C07295=1140.196,8.392,-49.288,179.724,6.289,149.221
C07296=1140.191,8.641,-49.301,179.727,6.291,149.220
C07297=1140.186,8.891,-49.315,179.729,6.291,149.220
C07298=1140.180,9.141,-49.329,179.732,6.292,149.219
C07299=1140.176,9.390,-49.342,179.734,6.293,149.219
C07300=1140.170,9.640,-49.355,179.737,6.294,149.218
C07301=1140.165,9.889,-49.370,179.739,6.295,149.218
C07302=1140.160,10.139,-49.382,179.741,6.296,149.217
C07303=1140.155,10.388,-49.397,179.744,6.296,149.216
C07304=1140.150,10.639,-49.410,179.747,6.298,149.216
C07305=1140.145,10.887,-49.423,179.749,6.298,149.215
C07306=1140.140,11.137,-49.438,179.752,6.299,149.215
C07307=1140.134,11.387,-49.451,179.754,6.300,149.214
C07308=1140.129,11.636,-49.465,179.757,6.301,149.214
C07309=1140.125,11.886,-49.478,179.759,6.302,149.213
C07310=1140.119,12.136,-49.492,179.762,6.303,149.213
C07311=1140.114,12.385,-49.506,179.765,6.304,149.212
C07312=1140.109,12.635,-49.520,179.767,6.305,149.212
C07313=1140.104,12.884,-49.533,179.770,6.305,149.211
C07314=1140.099,13.134,-49.547,179.772,6.306,149.210
C07315=1140.094,13.384,-49.561,179.775,6.307,149.210
C07316=1140.089,13.633,-49.575,179.777,6.308,149.209
C07317=1140.084,13.882,-49.588,179.779,6.309,149.209
C07318=1140.078,14.132,-49.602,179.782,6.310,149.208
C07319=1140.074,14.382,-49.616,179.785,6.311,149.208
C07320=1140.068,14.631,-49.630,179.787,6.312,149.207
C07321=1140.063,14.881,-49.644,179.790,6.312,149.207
C07322=1140.058,15.131,-49.657,179.792,6.314,149.206
C07323=1140.053,15.380,-49.671,179.795,6.314,149.206
C07324=1140.048,15.629,-49.685,179.797,6.315,149.205
C07325=1140.042,15.878,-49.699,179.800,6.316,149.204
C07326=1140.037,16.129,-49.713,179.802,6.317,149.204
C07327=1140.033,16.378,-49.727,179.805,6.318,149.203
C07328=1140.027,16.627,-49.741,179.808,6.319,149.203
C07329=1140.022,16.877,-49.755,179.810,6.320,149.202
C07330=1140.017,17.127,-49.769,179.812,6.321,149.202
C07331=1140.012,17.377,-49.783,179.815,6.322,149.201
C07332=1140.007,17.626,-49.797,179.818,6.323,149.201
C07333=1140.002,17.876,-49.811,179.820,6.323,149.200
C07334=1139.997,18.125,-49.825,179.823,6.325,149.199
C07335=1139.992,18.374,-49.838,179.825,6.326,149.199
C07336=1139.987,18.624,-49.853,179.828,6.326,149.199
C07337=1139.982,18.874,-49.866,179.830,6.327,149.198
C07338=1139.976,19.123,-49.880,179.833,6.328,149.197
C07339=1139.971,19.373,-49.894,179.835,6.329,149.197
C07340=1139.966,19.623,-49.909,179.838,6.330,149.196
C07341=1139.961,19.872,-49.923,179.841,6.331,149.196
C07342=1139.956,20.121,-49.937,179.843,6.332,149.195
C07343=1139.951,20.371,-49.951,179.845,6.333,149.195
C07344=1139.946,20.621,-49.965,179.848,6.334,149.194
C07345=1139.940,20.870,-49.979,179.851,6.335,149.194
C07346=1139.935,21.119,-49.994,179.854,6.336,149.193
C07347=1139.930,21.369,-50.008,179.856,6.337,149.193
C07348=1139.925,21.619,-50.022,179.858,6.337,149.192
C07349=1139.920,21.869,-50.037,179.861,6.339,149.191
C07350=1139.915,22.118,-50.050,179.864,6.340,149.191
C07351=1139.910,22.367,-50.065,179.866,6.340,149.190
C07352=1139.905,22.617,-50.079,179.869,6.342,149.190
C07353=1139.900,22.867,-50.093,179.871,6.342,149.189
C07354=1139.894,23.116,-50.107,179.874,6.343,149.189
C07355=1139.890,23.365,-50.121,179.876,6.345,149.188
C07356=1139.885,23.615,-50.136,179.879,6.345,149.188
C07357=1139.880,23.865,-50.150,179.881,6.346,149.187
C07358=1139.875,24.115,-50.164,179.884,6.347,149.186
C07359=1139.869,24.364,-50.178,179.887,6.348,149.186
C07360=1139.864,24.613,-50.192,179.889,6.349,149.186
C07361=1139.859,24.863,-50.207,179.892,6.350,149.185
C07362=1139.854,25.113,-50.221,179.894,6.351,149.184
C07363=1139.849,25.362,-50.235,179.897,6.353,149.184
C07364=1139.844,25.611,-50.249,179.900,6.353,149.183
C07365=1139.839,25.861,-50.264,179.902,6.354,149.183
C07366=1139.834,26.110,-50.278,179.905,6.355,149.182
C07367=1139.829,26.360,-50.293,179.907,6.356,149.182
C07368=1139.824,26.610,-50.307,179.909,6.357,149.181
C07369=1139.819,26.859,-50.321,179.913,6.358,149.181
C07370=1139.813,27.128,-50.337,179.915,6.359,149.180
C07371=1139.807,27.397,-50.352,179.918,6.360,149.179
C07372=1139.802,27.666,-50.368,179.921,6.362,149.179
C07373=1139.797,27.935,-50.384,179.923,6.362,149.178
C07374=1139.791,28.185,-50.399,179.926,6.363,149.178
C07375=1139.786,28.435,-50.413,179.929,6.364,149.177
C07376=1139.782,28.684,-50.427,179.931,6.365,149.177
C07377=1139.777,28.933,-50.442,179.934,6.367,149.176
C07378=1139.771,29.182,-50.456,179.936,6.367,149.176
C07379=1139.766,29.432,-50.470,179.939,6.368,149.175
C07380=1139.761,29.682,-50.485,179.941,6.370,149.175
C07381=1139.756,29.931,-50.500,179.944,6.370,149.174
C07382=1139.751,30.181,-50.514,179.947,6.372,149.174
C07383=1139.746,30.431,-50.529,179.949,6.373,149.173
C07384=1139.741,30.680,-50.544,179.952,6.373,149.172
C07385=1139.737,30.929,-50.558,179.954,6.375,149.172
C07386=1139.731,31.179,-50.573,179.957,6.375,149.171
C07387=1139.726,31.428,-50.588,179.960,6.377,149.171
C07388=1139.721,31.678,-50.602,179.962,6.378,149.170
C07389=1139.716,31.927,-50.616,179.965,6.379,149.170
C07390=1139.710,32.177,-50.632,179.967,6.380,149.169
C07391=1139.705,32.426,-50.646,179.969,6.380,149.169
C07392=1139.700,32.676,-50.660,179.973,6.382,149.168
C07393=1139.696,32.925,-50.675,179.975,6.383,149.168
C07394=1139.690,33.175,-50.690,179.978,6.384,149.167
C07395=1139.685,33.424,-50.705,179.980,6.385,149.167
C07396=1139.680,33.674,-50.719,179.982,6.385,149.166
C07397=1139.675,33.924,-50.734,179.986,6.387,149.165
C07398=1139.670,34.173,-50.749,179.988,6.387,149.165
C07399=1139.665,34.423,-50.763,179.991,6.389,149.165
C07400=1139.660,34.672,-50.778,179.993,6.390,149.164
C07401=1139.655,34.922,-50.793,179.996,6.391,149.163
C07402=1139.650,35.171,-50.808,179.998,6.392,149.163
C07403=1139.645,35.421,-50.823,-179.999,6.393,149.162
C07404=1139.640,35.670,-50.838,-179.996,6.394,149.162
C07405=1139.635,35.920,-50.852,-179.994,6.395,149.161
C07406=1139.630,36.169,-50.867,-179.991,6.396,149.161
C07407=1139.624,36.419,-50.882,-179.989,6.397,149.160
C07408=1139.620,36.668,-50.897,-179.986,6.399,149.160
C07409=1139.614,36.918,-50.912,-179.983,6.399,149.159
C07410=1139.609,37.167,-50.927,-179.981,6.401,149.159
C07411=1139.605,37.417,-50.941,-179.978,6.401,149.158
C07412=1139.599,37.666,-50.957,-179.975,6.403,149.158
C07413=1139.594,37.916,-50.971,-179.973,6.404,149.157
C07414=1139.589,38.165,-50.987,-179.970,6.404,149.156
C07415=1139.584,38.414,-51.002,-179.968,6.406,149.156
C07416=1139.579,38.664,-51.016,-179.965,6.407,149.156
C07417=1139.574,38.914,-51.032,-179.962,6.408,149.155
C07418=1139.569,39.163,-51.046,-179.960,6.409,149.154
C07419=1139.563,39.413,-51.062,-179.957,6.410,149.154
C07420=1139.559,39.662,-51.077,-179.955,6.411,149.153
C07421=1139.553,39.912,-51.091,-179.952,6.412,149.153
C07422=1139.549,40.162,-51.107,-179.950,6.413,149.152
C07423=1139.544,40.411,-51.122,-179.947,6.414,149.152
C07424=1139.539,40.661,-51.137,-179.944,6.415,149.151
C07425=1139.534,40.910,-51.152,-179.942,6.417,149.151
C07426=1139.529,41.159,-51.167,-179.939,6.417,149.150
C07427=1139.524,41.409,-51.182,-179.936,6.419,149.150
C07428=1139.518,41.658,-51.197,-179.934,6.420,149.149
C07429=1139.514,41.907,-51.212,-179.931,6.421,149.149
C07430=1139.508,42.157,-51.228,-179.929,6.422,149.148
C07431=1139.503,42.406,-51.242,-179.926,6.424,149.148
C07432=1139.498,42.656,-51.258,-179.923,6.424,149.147
C07433=1139.494,42.906,-51.273,-179.920,6.426,149.147
C07434=1139.489,43.155,-51.289,-179.918,6.426,149.146
C07435=1139.483,43.405,-51.303,-179.915,6.428,149.145
C07436=1139.478,43.654,-51.318,-179.913,6.429,149.145
C07437=1139.473,43.904,-51.334,-179.910,6.430,149.144
C07438=1139.468,44.153,-51.349,-179.907,6.431,149.144
C07439=1139.463,44.402,-51.365,-179.905,6.432,149.143
C07440=1139.459,44.652,-51.380,-179.902,6.433,149.143
C07441=1139.453,44.902,-51.395,-179.899,6.434,149.142
C07442=1139.448,45.151,-51.410,-179.897,6.435,149.142
C07443=1139.443,45.400,-51.425,-179.894,6.436,149.141
C07444=1139.438,45.650,-51.441,-179.892,6.437,149.141
C07445=1139.433,45.899,-51.456,-179.889,6.439,149.140
C07446=1139.428,46.149,-51.472,-179.886,6.439,149.140
C07447=1139.423,46.398,-51.487,-179.884,6.441,149.139
C07448=1139.418,46.647,-51.502,-179.881,6.442,149.139
C07449=1139.412,46.897,-51.517,-179.878,6.443,149.138
C07450=1139.408,47.147,-51.532,-179.876,6.444,149.138
C07451=1139.403,47.397,-51.548,-179.873,6.446,149.137
C07452=1139.398,47.646,-51.564,-179.871,6.446,149.136
C07453=1139.393,47.895,-51.579,-179.868,6.448,149.136
C07454=1139.388,48.145,-51.594,-179.866,6.449,149.136
C07455=1139.383,48.395,-51.610,-179.862,6.450,149.135
C07456=1139.378,48.644,-51.625,-179.860,6.451,149.134
C07457=1139.373,48.893,-51.641,-179.858,6.452,149.134
C07458=1139.367,49.143,-51.657,-179.855,6.453,149.134
C07459=1139.363,49.392,-51.672,-179.852,6.454,149.133
C07460=1139.358,49.642,-51.688,-179.849,6.456,149.132
C07461=1139.353,49.891,-51.703,-179.847,6.457,149.132
C07462=1139.347,50.141,-51.719,-179.844,6.458,149.131
C07463=1139.343,50.390,-51.734,-179.842,6.459,149.131
C07464=1139.338,50.640,-51.750,-179.839,6.461,149.130
C07465=1139.333,50.889,-51.766,-179.836,6.461,149.130
C07466=1139.327,51.138,-51.782,-179.834,6.463,149.129
C07467=1139.323,51.388,-51.797,-179.832,6.464,149.129
C07468=1139.318,51.637,-51.812,-179.828,6.465,149.128
C07469=1139.312,51.887,-51.828,-179.826,6.466,149.128
C07470=1139.307,52.136,-51.844,-179.823,6.467,149.127
C07471=1139.303,52.386,-51.859,-179.820,6.469,149.127
C07472=1139.298,52.635,-51.875,-179.818,6.469,149.126
C07473=1139.292,52.885,-51.890,-179.815,6.471,149.126
C07474=1139.287,53.153,-51.907,-179.813,6.472,149.125
C07475=1139.282,53.422,-51.925,-179.810,6.473,149.125
C07476=1139.276,53.691,-51.942,-179.807,6.474,149.124
C07477=1139.271,53.959,-51.958,-179.804,6.476,149.124
C07478=1139.266,54.208,-51.974,-179.801,6.477,149.123
C07479=1139.261,54.458,-51.990,-179.798,6.478,149.122
C07480=1139.256,54.707,-52.006,-179.796,6.479,149.122
C07481=1139.251,54.957,-52.021,-179.793,6.480,149.121
C07482=1139.246,55.207,-52.037,-179.790,6.482,149.121
C07483=1139.241,55.456,-52.053,-179.788,6.483,149.120
C07484=1139.235,55.705,-52.069,-179.785,6.484,149.120
C07485=1139.231,55.955,-52.085,-179.783,6.485,149.119
C07486=1139.226,56.204,-52.100,-179.780,6.487,149.119
C07487=1139.221,56.453,-52.117,-179.777,6.488,149.119
C07488=1139.216,56.703,-52.133,-179.775,6.489,149.118
C07489=1139.211,56.952,-52.148,-179.772,6.490,149.117
C07490=1139.206,57.202,-52.164,-179.770,6.491,149.117
C07491=1139.201,57.451,-52.180,-179.766,6.492,149.116
C07492=1139.196,57.701,-52.196,-179.764,6.494,149.116
C07493=1139.191,57.951,-52.212,-179.762,6.495,149.115
C07494=1139.186,58.200,-52.228,-179.758,6.496,149.115
C07495=1139.180,58.449,-52.244,-179.756,6.497,149.114
C07496=1139.176,58.698,-52.260,-179.753,6.499,149.114
C07497=1139.170,58.948,-52.276,-179.751,6.500,149.113
C07498=1139.166,59.198,-52.292,-179.748,6.501,149.113
C07499=1139.161,59.446,-52.308,-179.745,6.502,149.112
C07500=1139.156,59.696,-52.324,-179.743,6.503,149.112
C07501=1139.151,59.945,-52.340,-179.740,6.505,149.111
C07502=1139.146,60.195,-52.356,-179.737,6.506,149.111
C07503=1139.142,60.444,-52.372,-179.735,6.507,149.110
C07504=1139.136,60.694,-52.388,-179.732,6.508,149.110
C07505=1139.131,60.944,-52.404,-179.729,6.510,149.109
C07506=1139.126,61.193,-52.421,-179.727,6.511,149.109
C07507=1139.121,61.443,-52.437,-179.724,6.512,149.108
C07508=1139.116,61.692,-52.453,-179.721,6.513,149.108
C07509=1139.111,61.942,-52.469,-179.719,6.515,149.107
C07510=1139.106,62.191,-52.485,-179.716,6.516,149.107
C07511=1139.101,62.441,-52.501,-179.713,6.517,149.106
C07512=1139.096,62.689,-52.517,-179.711,6.518,149.106
C07513=1139.091,62.939,-52.534,-179.708,6.520,149.105
C07514=1139.086,63.188,-52.550,-179.706,6.521,149.105
C07515=1139.082,63.438,-52.566,-179.702,6.522,149.104
C07516=1139.076,63.687,-52.582,-179.700,6.523,149.104
C07517=1139.072,63.937,-52.599,-179.697,6.525,149.103
C07518=1139.066,64.186,-52.614,-179.694,6.526,149.103
C07519=1139.062,64.436,-52.631,-179.692,6.527,149.102
C07520=1139.056,64.685,-52.648,-179.689,6.528,149.102
C07521=1139.051,64.935,-52.664,-179.687,6.530,149.101
C07522=1139.046,65.184,-52.680,-179.684,6.530,149.101
C07523=1139.042,65.433,-52.697,-179.681,6.532,149.100
C07524=1139.036,65.682,-52.712,-179.678,6.534,149.100
C07525=1139.032,65.932,-52.729,-179.676,6.534,149.099
C07526=1139.027,66.181,-52.745,-179.673,6.536,149.099
C07527=1139.021,66.431,-52.762,-179.670,6.538,149.098
C07528=1139.016,66.680,-52.778,-179.668,6.538,149.098
C07529=1139.012,66.929,-52.795,-179.665,6.540,149.097
C07530=1139.007,67.179,-52.811,-179.662,6.541,149.097
C07531=1139.002,67.428,-52.827,-179.660,6.542,149.096
C07532=1138.997,67.678,-52.844,-179.657,6.544,149.096
C07533=1138.992,67.927,-52.861,-179.654,6.545,149.095
C07534=1138.987,68.177,-52.877,-179.652,6.546,149.095
C07535=1138.982,68.426,-52.893,-179.649,6.548,149.094
C07536=1138.977,68.675,-52.910,-179.646,6.549,149.094
C07537=1138.972,68.925,-52.927,-179.644,6.550,149.093
C07538=1138.967,69.174,-52.943,-179.641,6.551,149.093
C07539=1138.962,69.424,-52.959,-179.638,6.553,149.092
C07540=1138.957,69.673,-52.975,-179.636,6.553,149.092
C07541=1138.952,69.922,-52.993,-179.633,6.555,149.091
C07542=1138.947,70.172,-53.009,-179.630,6.557,149.091
C07543=1138.942,70.421,-53.026,-179.627,6.558,149.090
C07544=1138.938,70.670,-53.042,-179.625,6.559,149.090
C07545=1138.933,70.920,-53.060,-179.622,6.561,149.089
C07546=1138.927,71.169,-53.075,-179.619,6.562,149.089
C07547=1138.923,71.419,-53.092,-179.617,6.563,149.088
C07548=1138.917,71.669,-53.109,-179.614,6.564,149.088
C07549=1138.912,71.917,-53.125,-179.611,6.566,149.087
C07550=1138.908,72.167,-53.142,-179.609,6.567,149.087
C07551=1138.902,72.416,-53.159,-179.606,6.569,149.087
C07552=1138.898,72.666,-53.176,-179.603,6.570,149.086
C07553=1138.893,72.915,-53.192,-179.600,6.571,149.085
C07554=1138.887,73.164,-53.209,-179.598,6.572,149.085
C07555=1138.883,73.414,-53.226,-179.595,6.574,149.085
C07556=1138.878,73.663,-53.242,-179.592,6.575,149.084
C07557=1138.873,73.913,-53.260,-179.590,6.576,149.083
C07558=1138.868,74.162,-53.276,-179.587,6.578,149.083
C07559=1138.863,74.411,-53.293,-179.584,6.579,149.082
C07560=1138.858,74.661,-53.310,-179.581,6.581,149.082
C07561=1138.853,74.910,-53.326,-179.579,6.582,149.082
C07562=1138.848,75.160,-53.344,-179.576,6.583,149.081
C07563=1138.844,75.409,-53.360,-179.574,6.585,149.081
C07564=1138.838,75.659,-53.377,-179.571,6.585,149.080
C07565=1138.833,75.908,-53.394,-179.568,6.587,149.080
C07566=1138.828,76.157,-53.411,-179.566,6.589,149.079
C07567=1138.824,76.407,-53.428,-179.563,6.590,149.079
C07568=1138.818,76.656,-53.445,-179.560,6.591,149.078
C07569=1138.814,76.905,-53.462,-179.557,6.592,149.078
C07570=1138.809,77.154,-53.479,-179.555,6.594,149.077
C07571=1138.804,77.404,-53.496,-179.552,6.596,149.077
C07572=1138.799,77.653,-53.512,-179.549,6.596,149.076
C07573=1138.794,77.903,-53.530,-179.547,6.598,149.076
C07574=1138.789,78.152,-53.546,-179.544,6.600,149.075
C07575=1138.784,78.402,-53.563,-179.541,6.601,149.075
C07576=1138.780,78.651,-53.581,-179.538,6.602,149.074
C07577=1138.774,78.900,-53.598,-179.536,6.603,149.074
C07578=1138.768,79.169,-53.616,-179.533,6.605,149.073
C07579=1138.763,79.437,-53.634,-179.530,6.606,149.073
C07580=1138.758,79.706,-53.653,-179.527,6.608,149.072
C07581=1138.753,79.974,-53.671,-179.524,6.610,149.072
C07582=1138.748,80.224,-53.688,-179.521,6.611,149.071
C07583=1138.742,80.472,-53.706,-179.518,6.613,149.071
C07584=1138.738,80.722,-53.723,-179.516,6.613,149.070
C07585=1138.733,80.972,-53.740,-179.513,6.615,149.070
C07586=1138.729,81.220,-53.757,-179.510,6.616,149.069
C07587=1138.723,81.470,-53.774,-179.507,6.618,149.069
C07588=1138.718,81.719,-53.791,-179.505,6.619,149.068
C07589=1138.713,81.968,-53.809,-179.502,6.621,149.068
C07590=1138.708,82.218,-53.826,-179.500,6.622,149.068
C07591=1138.704,82.468,-53.843,-179.497,6.624,149.067
C07592=1138.699,82.717,-53.861,-179.494,6.625,149.066
C07593=1138.694,82.966,-53.878,-179.492,6.626,149.066
C07594=1138.689,83.216,-53.895,-179.489,6.628,149.066
C07595=1138.684,83.464,-53.912,-179.486,6.629,149.065
C07596=1138.678,83.714,-53.929,-179.483,6.631,149.065
C07597=1138.674,83.963,-53.947,-179.480,6.632,149.064
C07598=1138.669,84.213,-53.964,-179.478,6.633,149.064
C07599=1138.664,84.463,-53.981,-179.475,6.635,149.063
C07600=1138.660,84.712,-53.999,-179.472,6.636,149.063
C07601=1138.654,84.961,-54.016,-179.469,6.638,149.062
C07602=1138.649,85.211,-54.034,-179.467,6.639,149.062
C07603=1138.645,85.460,-54.051,-179.464,6.640,149.061
C07604=1138.639,85.708,-54.068,-179.462,6.642,149.061
C07605=1138.634,85.958,-54.086,-179.458,6.643,149.060
C07606=1138.629,86.207,-54.103,-179.456,6.645,149.060
C07607=1138.625,86.457,-54.120,-179.453,6.647,149.059
C07608=1138.620,86.706,-54.138,-179.451,6.647,149.059
C07609=1138.615,86.956,-54.155,-179.448,6.649,149.059
C07610=1138.610,87.205,-54.173,-179.445,6.650,149.058
C07611=1138.605,87.455,-54.190,-179.442,6.652,149.057
C07612=1138.600,87.704,-54.208,-179.439,6.654,149.057
C07613=1138.595,87.953,-54.226,-179.437,6.655,149.057
C07614=1138.590,88.203,-54.243,-179.434,6.656,149.056
C07615=1138.585,88.452,-54.261,-179.431,6.658,149.056
C07616=1138.581,88.701,-54.278,-179.429,6.659,149.055
C07617=1138.576,88.951,-54.296,-179.426,6.661,149.055
C07618=1138.571,89.200,-54.314,-179.423,6.663,149.054
C07619=1138.566,89.450,-54.331,-179.421,6.663,149.054
C07620=1138.561,89.699,-54.349,-179.418,6.665,149.053
C07621=1138.557,89.948,-54.367,-179.415,6.666,149.053
C07622=1138.552,90.197,-54.384,-179.412,6.668,149.052
C07623=1138.547,90.447,-54.402,-179.409,6.670,149.052
C07624=1138.542,90.696,-54.420,-179.407,6.671,149.052
C07625=1138.536,90.946,-54.437,-179.404,6.673,149.051
C07626=1138.532,91.195,-54.455,-179.401,6.674,149.050
C07627=1138.527,91.444,-54.473,-179.399,6.675,149.050
C07628=1138.522,91.693,-54.491,-179.396,6.677,149.050
C07629=1138.517,91.943,-54.508,-179.393,6.679,149.049
C07630=1138.512,92.192,-54.526,-179.390,6.680,149.049
C07631=1138.507,92.441,-54.544,-179.388,6.682,149.048
C07632=1138.503,92.690,-54.562,-179.385,6.682,149.048
C07633=1138.497,92.940,-54.579,-179.382,6.684,149.047
C07634=1138.492,93.189,-54.597,-179.380,6.686,149.047
C07635=1138.487,93.438,-54.615,-179.377,6.687,149.046
C07636=1138.483,93.687,-54.633,-179.374,6.689,149.046
C07637=1138.478,93.937,-54.651,-179.371,6.691,149.046
C07638=1138.473,94.186,-54.669,-179.368,6.692,149.045
C07639=1138.468,94.436,-54.686,-179.365,6.694,149.045
C07640=1138.463,94.685,-54.704,-179.363,6.695,149.044
C07641=1138.458,94.935,-54.722,-179.361,6.696,149.044
C07642=1138.453,95.184,-54.740,-179.358,6.698,149.043
C07643=1138.448,95.433,-54.758,-179.355,6.700,149.043
C07644=1138.444,95.682,-54.776,-179.352,6.701,149.042
C07645=1138.439,95.931,-54.794,-179.349,6.703,149.042
C07646=1138.434,96.180,-54.812,-179.346,6.704,149.041
C07647=1138.429,96.430,-54.830,-179.344,6.706,149.041
C07648=1138.424,96.679,-54.848,-179.341,6.708,149.041
C07649=1138.419,96.928,-54.866,-179.339,6.708,149.040
C07650=1138.415,97.178,-54.884,-179.336,6.710,149.039
C07651=1138.410,97.427,-54.902,-179.333,6.711,149.039
C07652=1138.405,97.676,-54.920,-179.330,6.713,149.039
C07653=1138.400,97.925,-54.938,-179.327,6.715,149.038
C07654=1138.395,98.175,-54.956,-179.325,6.716,149.038
C07655=1138.390,98.424,-54.974,-179.322,6.718,149.037
C07656=1138.384,98.673,-54.993,-179.319,6.720,149.037
C07657=1138.380,98.923,-55.011,-179.316,6.721,149.036
C07658=1138.375,99.172,-55.029,-179.313,6.723,149.036
C07659=1138.370,99.421,-55.047,-179.311,6.724,149.036
C07660=1138.365,99.671,-55.065,-179.308,6.725,149.035
C07661=1138.361,99.920,-55.083,-179.306,6.727,149.035
C07662=1138.356,100.169,-55.101,-179.303,6.729,149.034
C07663=1138.351,100.419,-55.120,-179.300,6.730,149.034
C07664=1138.346,100.668,-55.138,-179.297,6.732,149.033
C07665=1138.341,100.918,-55.156,-179.294,6.733,149.033
C07666=1138.336,101.166,-55.175,-179.291,6.735,149.032
C07667=1138.331,101.415,-55.193,-179.289,6.737,149.032
C07668=1138.327,101.665,-55.211,-179.286,6.738,149.032
C07669=1138.321,101.915,-55.230,-179.283,6.740,149.031
C07670=1138.316,102.164,-55.248,-179.280,6.742,149.031
C07671=1138.311,102.413,-55.266,-179.278,6.743,149.030
C07672=1138.307,102.662,-55.285,-179.275,6.744,149.030
C07673=1138.303,102.911,-55.303,-179.272,6.746,149.029
C07674=1138.297,103.161,-55.321,-179.270,6.747,149.029
C07675=1138.292,103.410,-55.339,-179.267,6.749,149.028
C07676=1138.288,103.659,-55.358,-179.264,6.751,149.028
C07677=1138.283,103.908,-55.376,-179.261,6.752,149.028
C07678=1138.277,104.158,-55.395,-179.259,6.754,149.027
C07679=1138.272,104.407,-55.413,-179.256,6.756,149.027
C07680=1138.268,104.656,-55.432,-179.253,6.757,149.026
C07681=1138.264,104.906,-55.450,-179.250,6.759,149.026
C07682=1138.258,105.174,-55.470,-179.247,6.760,149.025
C07683=1138.253,105.442,-55.490,-179.245,6.762,149.025
C07684=1138.248,105.711,-55.510,-179.241,6.764,149.024
C07685=1138.243,105.979,-55.530,-179.238,6.766,149.024
C07686=1138.237,106.229,-55.548,-179.235,6.767,149.023
C07687=1138.232,106.477,-55.567,-179.232,6.769,149.023
C07688=1138.228,106.727,-55.585,-179.230,6.771,149.023
C07689=1138.223,106.976,-55.605,-179.227,6.772,149.022
C07690=1138.218,107.225,-55.623,-179.224,6.774,149.022
C07691=1138.214,107.475,-55.641,-179.222,6.776,149.021
C07692=1138.208,107.724,-55.660,-179.219,6.777,149.021
C07693=1138.203,107.973,-55.678,-179.217,6.778,149.021
C07694=1138.199,108.222,-55.697,-179.213,6.780,149.020
C07695=1138.194,108.472,-55.716,-179.211,6.781,149.020
C07696=1138.189,108.720,-55.735,-179.208,6.783,149.019
C07697=1138.184,108.971,-55.754,-179.205,6.785,149.019
C07698=1138.179,109.219,-55.772,-179.203,6.786,149.018
C07699=1138.174,109.469,-55.791,-179.200,6.788,149.018
C07700=1138.170,109.718,-55.810,-179.197,6.790,149.017
C07701=1138.165,109.967,-55.828,-179.194,6.791,149.017
C07702=1138.160,110.217,-55.848,-179.192,6.793,149.017
C07703=1138.155,110.466,-55.866,-179.189,6.795,149.016
C07704=1138.150,110.715,-55.885,-179.186,6.796,149.016
C07705=1138.146,110.964,-55.904,-179.183,6.798,149.015
C07706=1138.140,111.214,-55.922,-179.180,6.799,149.015
C07707=1138.136,111.463,-55.942,-179.177,6.801,149.014
C07708=1138.130,111.712,-55.960,-179.175,6.803,149.014
C07709=1138.126,111.961,-55.979,-179.172,6.805,149.014
C07710=1138.121,112.210,-55.998,-179.169,6.806,149.013
C07711=1138.116,112.460,-56.016,-179.167,6.808,149.013
C07712=1138.111,112.709,-56.036,-179.164,6.810,149.012
C07713=1138.107,112.958,-56.055,-179.161,6.811,149.012
C07714=1138.102,113.208,-56.074,-179.158,6.813,149.012
C07715=1138.097,113.456,-56.092,-179.156,6.815,149.011
C07716=1138.092,113.705,-56.112,-179.153,6.816,149.011
C07717=1138.088,113.955,-56.130,-179.150,6.819,149.010
C07718=1138.082,114.204,-56.149,-179.147,6.820,149.010
C07719=1138.077,114.454,-56.169,-179.144,6.822,149.010
C07720=1138.073,114.703,-56.187,-179.141,6.823,149.009
C07721=1138.068,114.952,-56.207,-179.138,6.825,149.008
C07722=1138.063,115.201,-56.225,-179.135,6.827,149.008
C07723=1138.058,115.450,-56.245,-179.133,6.829,149.008
C07724=1138.053,115.699,-56.264,-179.130,6.830,149.007
C07725=1138.049,115.949,-56.283,-179.127,6.832,149.007
C07726=1138.043,116.198,-56.302,-179.125,6.834,149.006
C07727=1138.039,116.448,-56.322,-179.122,6.835,149.006
C07728=1138.034,116.696,-56.340,-179.119,6.837,149.006
C07729=1138.029,116.946,-56.360,-179.116,6.839,149.005
C07730=1138.024,117.195,-56.378,-179.114,6.840,149.005
C07731=1138.020,117.445,-56.398,-179.111,6.842,149.004
C07732=1138.014,117.693,-56.417,-179.108,6.844,149.004
C07733=1138.010,117.943,-56.436,-179.105,6.845,149.004
C07734=1138.005,118.191,-56.455,-179.103,6.847,149.003
C07735=1138.000,118.441,-56.475,-179.100,6.849,149.003
C07736=1137.996,118.691,-56.495,-179.097,6.850,149.002
C07737=1137.991,118.939,-56.513,-179.095,6.852,149.002
C07738=1137.986,119.189,-56.533,-179.092,6.854,149.002
C07739=1137.981,119.438,-56.552,-179.088,6.856,149.001
C07740=1137.976,119.687,-56.572,-179.086,6.858,149.001
C07741=1137.972,119.936,-56.591,-179.083,6.860,149.000
C07742=1137.967,120.185,-56.610,-179.080,6.861,149.000
C07743=1137.962,120.435,-56.630,-179.078,6.863,149.000
C07744=1137.957,120.684,-56.649,-179.075,6.865,148.999
C07745=1137.953,120.933,-56.668,-179.072,6.866,148.999
C07746=1137.947,121.182,-56.687,-179.069,6.868,148.998
C07747=1137.943,121.431,-56.707,-179.066,6.869,148.998
C07748=1137.938,121.681,-56.727,-179.063,6.871,148.997
C07749=1137.933,121.930,-56.745,-179.061,6.873,148.997
C07750=1137.928,122.179,-56.765,-179.058,6.874,148.997
C07751=1137.923,122.428,-56.784,-179.055,6.876,148.996
C07752=1137.918,122.678,-56.804,-179.052,6.879,148.996
C07753=1137.914,122.927,-56.824,-179.049,6.880,148.995
C07754=1137.908,123.176,-56.843,-179.047,6.882,148.995
C07755=1137.905,123.425,-56.863,-179.044,6.884,148.995
C07756=1137.900,123.674,-56.882,-179.041,6.885,148.994
C07757=1137.895,123.923,-56.902,-179.038,6.887,148.994
C07758=1137.890,124.173,-56.921,-179.036,6.889,148.993
C07759=1137.885,124.422,-56.941,-179.033,6.890,148.993
C07760=1137.880,124.671,-56.960,-179.030,6.892,148.993
C07761=1137.875,124.920,-56.981,-179.027,6.894,148.992
C07762=1137.871,125.169,-57.000,-179.024,6.896,148.992
C07763=1137.866,125.418,-57.019,-179.021,6.898,148.991
C07764=1137.861,125.668,-57.039,-179.019,6.900,148.991
C07765=1137.857,125.917,-57.059,-179.016,6.901,148.991
C07766=1137.852,126.166,-57.079,-179.013,6.903,148.990
C07767=1137.847,126.415,-57.098,-179.010,6.905,148.990
C07768=1137.842,126.665,-57.118,-179.008,6.907,148.989
C07769=1137.837,126.914,-57.138,-179.005,6.908,148.989
C07770=1137.832,127.162,-57.157,-179.002,6.911,148.989
C07771=1137.827,127.412,-57.177,-178.999,6.912,148.988
C07772=1137.823,127.661,-57.197,-178.996,6.914,148.988
C07773=1137.818,127.911,-57.217,-178.994,6.916,148.988
C07774=1137.813,128.159,-57.236,-178.991,6.918,148.987
C07775=1137.808,128.408,-57.257,-178.989,6.920,148.987
C07776=1137.804,128.658,-57.276,-178.986,6.921,148.986
C07777=1137.799,128.908,-57.296,-178.983,6.924,148.986
C07778=1137.794,129.156,-57.316,-178.980,6.925,148.986
C07779=1137.789,129.405,-57.336,-178.977,6.927,148.985
C07780=1137.785,129.654,-57.356,-178.974,6.929,148.985
C07781=1137.780,129.904,-57.376,-178.972,6.930,148.984
C07782=1137.775,130.152,-57.396,-178.969,6.932,148.984
C07783=1137.770,130.402,-57.415,-178.966,6.934,148.984
C07784=1137.765,130.651,-57.435,-178.963,6.936,148.983
C07785=1137.761,130.900,-57.455,-178.960,6.938,148.983
C07786=1137.755,131.169,-57.477,-178.957,6.940,148.982
C07787=1137.751,131.437,-57.499,-178.954,6.942,148.982
C07788=1137.745,131.706,-57.521,-178.951,6.944,148.982
C07789=1137.740,131.975,-57.542,-178.948,6.945,148.981
C07790=1137.736,132.224,-57.562,-178.945,6.948,148.981
C07791=1137.730,132.473,-57.581,-178.943,6.950,148.980
C07792=1137.725,132.722,-57.602,-178.940,6.952,148.980
C07793=1137.720,132.971,-57.622,-178.937,6.953,148.980
C07794=1137.716,133.220,-57.642,-178.934,6.955,148.979
C07795=1137.712,133.469,-57.663,-178.932,6.957,148.979
C07796=1137.707,133.719,-57.682,-178.928,6.959,148.979
C07797=1137.702,133.967,-57.702,-178.926,6.961,148.978
C07798=1137.696,134.217,-57.723,-178.923,6.963,148.978
C07799=1137.692,134.466,-57.743,-178.920,6.964,148.977
C07800=1137.687,134.715,-57.763,-178.918,6.966,148.977
C07801=1137.683,134.965,-57.783,-178.914,6.968,148.977
C07802=1137.678,135.213,-57.803,-178.912,6.970,148.976
C07803=1137.673,135.463,-57.824,-178.909,6.972,148.976
C07804=1137.669,135.712,-57.845,-178.906,6.974,148.975
C07805=1137.663,135.961,-57.864,-178.904,6.976,148.975
C07806=1137.659,136.209,-57.884,-178.901,6.977,148.975
C07807=1137.654,136.459,-57.905,-178.898,6.980,148.974
C07808=1137.649,136.708,-57.925,-178.895,6.981,148.974
C07809=1137.645,136.957,-57.945,-178.892,6.983,148.974
C07810=1137.640,137.206,-57.966,-178.890,6.985,148.973
C07811=1137.635,137.455,-57.987,-178.886,6.987,148.973
C07812=1137.630,137.704,-58.007,-178.884,6.989,148.973
C07813=1137.626,137.954,-58.027,-178.881,6.991,148.972
C07814=1137.621,138.203,-58.048,-178.878,6.992,148.972
C07815=1137.616,138.452,-58.068,-178.875,6.994,148.971
C07816=1137.612,138.701,-58.088,-178.872,6.997,148.971
C07817=1137.607,138.950,-58.109,-178.870,6.999,148.971
C07818=1137.602,139.199,-58.130,-178.867,7.000,148.970
C07819=1137.597,139.449,-58.149,-178.864,7.002,148.970
C07820=1137.592,139.698,-58.170,-178.862,7.004,148.970
C07821=1137.588,139.947,-58.191,-178.858,7.006,148.969
C07822=1137.583,140.196,-58.211,-178.856,7.008,148.969
C07823=1137.578,140.445,-58.232,-178.853,7.010,148.968
C07824=1137.574,140.694,-58.252,-178.850,7.011,148.968
C07825=1137.569,140.943,-58.273,-178.847,7.014,148.968
C07826=1137.564,141.192,-58.294,-178.844,7.016,148.967
C07827=1137.560,141.441,-58.314,-178.842,7.018,148.967
C07828=1137.554,141.691,-58.335,-178.839,7.019,148.967
C07829=1137.550,141.940,-58.356,-178.836,7.022,148.966
C07830=1137.545,142.189,-58.376,-178.833,7.024,148.966
C07831=1137.540,142.438,-58.397,-178.831,7.025,148.966
C07832=1137.536,142.687,-58.417,-178.828,7.027,148.965
C07833=1137.531,142.936,-58.438,-178.825,7.030,148.965
C07834=1137.526,143.185,-58.459,-178.822,7.031,148.964
C07835=1137.521,143.434,-58.480,-178.820,7.033,148.964
C07836=1137.517,143.683,-58.500,-178.817,7.035,148.964
C07837=1137.512,143.932,-58.521,-178.814,7.038,148.963
C07838=1137.507,144.181,-58.541,-178.811,7.039,148.963
C07839=1137.502,144.431,-58.562,-178.808,7.041,148.963
C07840=1137.498,144.679,-58.583,-178.805,7.043,148.962
C07841=1137.493,144.928,-58.604,-178.802,7.045,148.962
C07842=1137.488,145.177,-58.625,-178.800,7.047,148.962
C07843=1137.484,145.427,-58.646,-178.797,7.049,148.961
C07844=1137.479,145.676,-58.666,-178.794,7.051,148.961
C07845=1137.474,145.925,-58.687,-178.791,7.053,148.961
C07846=1137.469,146.174,-58.709,-178.788,7.055,148.960
C07847=1137.465,146.423,-58.729,-178.786,7.057,148.960
C07848=1137.460,146.672,-58.750,-178.782,7.059,148.959
C07849=1137.455,146.921,-58.771,-178.780,7.061,148.959
C07850=1137.450,147.170,-58.792,-178.777,7.063,148.959
C07851=1137.445,147.419,-58.813,-178.774,7.065,148.959
C07852=1137.441,147.669,-58.834,-178.771,7.067,148.958
C07853=1137.436,147.918,-58.855,-178.769,7.069,148.958
C07854=1137.432,148.167,-58.875,-178.766,7.070,148.957
C07855=1137.427,148.416,-58.897,-178.763,7.073,148.957
C07856=1137.422,148.665,-58.918,-178.760,7.075,148.957
C07857=1137.417,148.914,-58.938,-178.758,7.077,148.956
C07858=1137.413,149.163,-58.961,-178.754,7.079,148.956
C07859=1137.408,149.412,-58.981,-178.752,7.081,148.956
C07860=1137.403,149.661,-59.002,-178.749,7.083,148.955
C07861=1137.398,149.910,-59.024,-178.746,7.085,148.955
C07862=1137.393,150.159,-59.044,-178.743,7.087,148.955
C07863=1137.389,150.408,-59.066,-178.741,7.089,148.954
C07864=1137.385,150.658,-59.087,-178.738,7.091,148.954
C07865=1137.379,150.907,-59.108,-178.735,7.093,148.954
C07866=1137.374,151.155,-59.130,-178.732,7.095,148.953
C07867=1137.370,151.404,-59.150,-178.730,7.097,148.953
C07868=1137.365,151.653,-59.172,-178.726,7.099,148.953
C07869=1137.361,151.903,-59.193,-178.724,7.101,148.952
C07870=1137.356,152.152,-59.215,-178.721,7.103,148.952
C07871=1137.351,152.401,-59.235,-178.718,7.105,148.952
C07872=1137.346,152.649,-59.257,-178.715,7.107,148.951
C07873=1137.342,152.899,-59.278,-178.713,7.109,148.951
C07874=1137.337,153.148,-59.300,-178.709,7.112,148.951
C07875=1137.332,153.397,-59.321,-178.707,7.113,148.950
C07876=1137.328,153.645,-59.342,-178.704,7.115,148.950
C07877=1137.323,153.895,-59.363,-178.701,7.118,148.950
C07878=1137.318,154.144,-59.385,-178.698,7.120,148.949
C07879=1137.313,154.393,-59.406,-178.696,7.121,148.949
C07880=1137.309,154.643,-59.428,-178.692,7.124,148.949
C07881=1137.304,154.891,-59.449,-178.690,7.126,148.949
C07882=1137.299,155.140,-59.470,-178.687,7.128,148.948
C07883=1137.295,155.389,-59.492,-178.684,7.130,148.948
C07884=1137.290,155.638,-59.514,-178.681,7.132,148.947
C07885=1137.285,155.887,-59.535,-178.678,7.134,148.947
C07886=1137.280,156.136,-59.556,-178.676,7.136,148.947
C07887=1137.276,156.385,-59.578,-178.673,7.138,148.946
C07888=1137.271,156.635,-59.599,-178.670,7.141,148.946
C07889=1137.266,156.883,-59.621,-178.667,7.142,148.946
C07890=1137.261,157.152,-59.644,-178.664,7.145,148.945
C07891=1137.256,157.421,-59.668,-178.661,7.147,148.945
C07892=1137.251,157.690,-59.691,-178.658,7.149,148.945
C07893=1137.246,157.960,-59.714,-178.655,7.152,148.945
C07894=1137.241,158.208,-59.736,-178.652,7.154,148.944
C07895=1137.237,158.458,-59.758,-178.650,7.155,148.944
C07896=1137.232,158.706,-59.779,-178.646,7.158,148.943
C07897=1137.227,158.956,-59.801,-178.644,7.160,148.943
C07898=1137.222,159.205,-59.822,-178.641,7.162,148.943
C07899=1137.218,159.453,-59.844,-178.638,7.164,148.942
C07900=1137.213,159.703,-59.866,-178.635,7.166,148.942
C07901=1137.208,159.951,-59.888,-178.633,7.169,148.942
C07902=1137.204,160.201,-59.910,-178.630,7.171,148.942
C07903=1137.199,160.449,-59.931,-178.627,7.172,148.941
C07904=1137.194,160.699,-59.952,-178.624,7.175,148.941
C07905=1137.190,160.948,-59.974,-178.622,7.177,148.941
C07906=1137.185,161.197,-59.996,-178.618,7.179,148.940
C07907=1137.181,161.446,-60.018,-178.616,7.181,148.940
C07908=1137.176,161.695,-60.040,-178.613,7.183,148.940
C07909=1137.172,161.944,-60.062,-178.610,7.186,148.939
C07910=1137.167,162.193,-60.084,-178.607,7.187,148.939
C07911=1137.162,162.441,-60.105,-178.604,7.190,148.939
C07912=1137.158,162.691,-60.127,-178.602,7.192,148.939
C07913=1137.153,162.939,-60.149,-178.599,7.194,148.938
C07914=1137.148,163.189,-60.171,-178.596,7.196,148.938
C07915=1137.144,163.437,-60.193,-178.593,7.198,148.937
C07916=1137.138,163.687,-60.215,-178.590,7.201,148.937
C07917=1137.134,163.935,-60.237,-178.588,7.203,148.937
C07918=1137.129,164.185,-60.259,-178.584,7.205,148.937
C07919=1137.124,164.433,-60.281,-178.582,7.207,148.936
C07920=1137.120,164.683,-60.303,-178.579,7.209,148.936
C07921=1137.115,164.931,-60.325,-178.576,7.211,148.936
C07922=1137.111,165.180,-60.347,-178.573,7.213,148.935
C07923=1137.106,165.429,-60.370,-178.570,7.216,148.935
C07924=1137.102,165.678,-60.392,-178.568,7.218,148.935
C07925=1137.097,165.927,-60.413,-178.564,7.220,148.934
C07926=1137.092,166.176,-60.435,-178.562,7.222,148.934
C07927=1137.087,166.425,-60.458,-178.560,7.224,148.934
C07928=1137.083,166.675,-60.480,-178.556,7.227,148.934
C07929=1137.078,166.923,-60.502,-178.554,7.229,148.933
C07930=1137.074,167.172,-60.524,-178.551,7.231,148.933
C07931=1137.068,167.421,-60.546,-178.548,7.233,148.933
C07932=1137.064,167.670,-60.568,-178.545,7.236,148.933
C07933=1137.060,167.919,-60.591,-178.542,7.237,148.932
C07934=1137.055,168.168,-60.613,-178.539,7.240,148.932
C07935=1137.050,168.417,-60.636,-178.537,7.242,148.932
C07936=1137.045,168.666,-60.657,-178.534,7.245,148.931
C07937=1137.041,168.915,-60.680,-178.531,7.246,148.931
C07938=1137.036,169.164,-60.702,-178.529,7.248,148.931
C07939=1137.031,169.413,-60.724,-178.525,7.251,148.930
C07940=1137.027,169.662,-60.747,-178.523,7.253,148.930
C07941=1137.022,169.911,-60.769,-178.520,7.255,148.930
C07942=1137.017,170.160,-60.791,-178.517,7.257,148.930
C07943=1137.013,170.408,-60.814,-178.514,7.260,148.929
C07944=1137.008,170.658,-60.836,-178.512,7.262,148.929
C07945=1137.004,170.907,-60.859,-178.508,7.264,148.929
C07946=1136.999,171.155,-60.881,-178.506,7.266,148.928
C07947=1136.994,171.405,-60.904,-178.503,7.269,148.928
C07948=1136.990,171.653,-60.926,-178.500,7.271,148.928
C07949=1136.984,171.902,-60.949,-178.497,7.273,148.927
C07950=1136.980,172.151,-60.971,-178.495,7.275,148.927
C07951=1136.976,172.400,-60.993,-178.491,7.278,148.927
C07952=1136.971,172.649,-61.016,-178.489,7.279,148.927
C07953=1136.967,172.898,-61.038,-178.486,7.282,148.926
C07954=1136.962,173.148,-61.061,-178.483,7.284,148.926
C07955=1136.957,173.396,-61.083,-178.480,7.287,148.926
C07956=1136.952,173.645,-61.107,-178.478,7.289,148.926
C07957=1136.948,173.894,-61.129,-178.474,7.291,148.925
C07958=1136.943,174.142,-61.152,-178.472,7.293,148.925
C07959=1136.939,174.392,-61.174,-178.469,7.296,148.925
C07960=1136.934,174.641,-61.197,-178.466,7.298,148.924
C07961=1136.929,174.890,-61.219,-178.463,7.300,148.924
C07962=1136.924,175.139,-61.242,-178.460,7.302,148.924
C07963=1136.920,175.387,-61.265,-178.458,7.305,148.924
C07964=1136.915,175.637,-61.288,-178.455,7.307,148.923
C07965=1136.911,175.885,-61.310,-178.452,7.309,148.923
C07966=1136.906,176.135,-61.333,-178.449,7.311,148.923
C07967=1136.902,176.383,-61.356,-178.446,7.314,148.923
C07968=1136.897,176.632,-61.379,-178.444,7.316,148.922
C07969=1136.893,176.880,-61.401,-178.441,7.318,148.922
C07970=1136.888,177.130,-61.424,-178.438,7.320,148.922
C07971=1136.883,177.379,-61.447,-178.435,7.323,148.922
C07972=1136.879,177.628,-61.470,-178.432,7.325,148.921
C07973=1136.873,177.877,-61.492,-178.430,7.328,148.921
C07974=1136.869,178.125,-61.515,-178.426,7.330,148.921
C07975=1136.865,178.374,-61.538,-178.424,7.332,148.920
C07976=1136.860,178.624,-61.562,-178.421,7.335,148.920
C07977=1136.855,178.872,-61.584,-178.418,7.337,148.920
C07978=1136.850,179.121,-61.607,-178.415,7.339,148.920
C07979=1136.846,179.370,-61.630,-178.413,7.341,148.919
C07980=1136.842,179.619,-61.653,-178.409,7.344,148.919
C07981=1136.837,179.868,-61.676,-178.407,7.346,148.919
C07982=1136.833,180.117,-61.699,-178.404,7.348,148.919
C07983=1136.827,180.366,-61.721,-178.401,7.350,148.918
C07984=1136.823,180.615,-61.745,-178.398,7.353,148.918
C07985=1136.818,180.864,-61.768,-178.395,7.356,148.918
C07986=1136.814,181.112,-61.791,-178.393,7.358,148.918
C07987=1136.809,181.361,-61.814,-178.390,7.360,148.917
C07988=1136.805,181.610,-61.838,-178.387,7.362,148.917
C07989=1136.800,181.859,-61.860,-178.384,7.365,148.917
C07990=1136.795,182.108,-61.883,-178.382,7.367,148.917
C07991=1136.791,182.357,-61.907,-178.378,7.369,148.916
C07992=1136.786,182.606,-61.930,-178.375,7.372,148.916
C07993=1136.782,182.854,-61.953,-178.373,7.374,148.916
C07994=1136.777,183.124,-61.978,-178.370,7.377,148.916
C07995=1136.771,183.394,-62.003,-178.367,7.379,148.915
C07996=1136.766,183.663,-62.029,-178.363,7.382,148.915
C07997=1136.762,183.933,-62.054,-178.361,7.385,148.915
C07998=1136.758,184.182,-62.077,-178.358,7.386,148.914
C07999=1136.752,184.431,-62.100,-178.355,7.389,148.914
C08000=1136.748,184.680,-62.123,-178.352,7.391,148.914
C08001=1136.743,184.929,-62.147,-178.349,7.394,148.914
C08002=1136.738,185.178,-62.170,-178.346,7.397,148.913
C08003=1136.734,185.427,-62.193,-178.344,7.398,148.913
C08004=1136.730,185.675,-62.216,-178.341,7.401,148.913
C08005=1136.725,185.924,-62.240,-178.338,7.403,148.913
C08006=1136.720,186.173,-62.263,-178.335,7.406,148.913
C08007=1136.716,186.422,-62.287,-178.332,7.408,148.912
C08008=1136.711,186.671,-62.310,-178.330,7.410,148.912
C08009=1136.706,186.920,-62.334,-178.326,7.413,148.912
C08010=1136.702,187.168,-62.358,-178.324,7.415,148.912
C08011=1136.697,187.417,-62.381,-178.321,7.418,148.911
C08012=1136.693,187.666,-62.404,-178.318,7.420,148.911
C08013=1136.688,187.915,-62.428,-178.315,7.422,148.911
C08014=1136.684,188.164,-62.452,-178.313,7.425,148.911
C08015=1136.679,188.413,-62.475,-178.310,7.427,148.910
C08016=1136.675,188.662,-62.498,-178.307,7.430,148.910
C08017=1136.670,188.911,-62.521,-178.304,7.432,148.910
C08018=1136.666,189.159,-62.545,-178.302,7.434,148.910
C08019=1136.661,189.408,-62.569,-178.298,7.437,148.909
C08020=1136.656,189.657,-62.592,-178.295,7.440,148.909
C08021=1136.652,189.906,-62.616,-178.293,7.441,148.909
C08022=1136.647,190.155,-62.640,-178.290,7.444,148.909
C08023=1136.642,190.404,-62.663,-178.287,7.447,148.908
C08024=1136.637,190.652,-62.687,-178.284,7.449,148.908
C08025=1136.633,190.901,-62.711,-178.282,7.452,148.908
C08026=1136.628,191.150,-62.735,-178.279,7.454,148.908
C08027=1136.624,191.399,-62.758,-178.276,7.456,148.908
C08028=1136.619,191.648,-62.782,-178.273,7.459,148.907
C08029=1136.615,191.896,-62.806,-178.271,7.461,148.907
C08030=1136.610,192.145,-62.829,-178.267,7.464,148.907
C08031=1136.605,192.394,-62.853,-178.264,7.467,148.907
C08032=1136.601,192.643,-62.876,-178.262,7.468,148.906
C08033=1136.597,192.892,-62.901,-178.259,7.471,148.906
C08034=1136.592,193.141,-62.924,-178.256,7.474,148.906
C08035=1136.587,193.390,-62.949,-178.253,7.476,148.906
C08036=1136.582,193.639,-62.972,-178.251,7.479,148.906
C08037=1136.578,193.887,-62.996,-178.247,7.481,148.905
C08038=1136.573,194.136,-63.020,-178.245,7.483,148.905
C08039=1136.569,194.384,-63.044,-178.242,7.486,148.905
C08040=1136.565,194.633,-63.068,-178.239,7.489,148.905
C08041=1136.560,194.883,-63.092,-178.236,7.490,148.904
C08042=1136.555,195.131,-63.116,-178.233,7.493,148.904
C08043=1136.551,195.380,-63.140,-178.230,7.496,148.904
C08044=1136.546,195.629,-63.164,-178.228,7.498,148.904
C08045=1136.542,195.877,-63.188,-178.225,7.501,148.904
C08046=1136.536,196.127,-63.212,-178.222,7.503,148.903
C08047=1136.532,196.375,-63.236,-178.220,7.505,148.903
C08048=1136.528,196.624,-63.260,-178.216,7.508,148.903
C08049=1136.524,196.872,-63.284,-178.214,7.511,148.903
C08050=1136.519,197.122,-63.308,-178.211,7.513,148.903
C08051=1136.514,197.370,-63.332,-178.208,7.516,148.902
C08052=1136.510,197.619,-63.356,-178.205,7.518,148.902
C08053=1136.506,197.868,-63.381,-178.202,7.521,148.902
C08054=1136.500,198.117,-63.405,-178.200,7.523,148.902
C08055=1136.496,198.366,-63.429,-178.197,7.526,148.902
C08056=1136.492,198.614,-63.453,-178.194,7.528,148.901
C08057=1136.487,198.862,-63.477,-178.191,7.531,148.901
C08058=1136.483,199.112,-63.502,-178.188,7.533,148.901
C08059=1136.478,199.361,-63.525,-178.185,7.536,148.901
C08060=1136.474,199.609,-63.550,-178.182,7.539,148.901
C08061=1136.468,199.858,-63.574,-178.180,7.541,148.900
C08062=1136.465,200.107,-63.599,-178.177,7.544,148.900
C08063=1136.460,200.355,-63.623,-178.174,7.546,148.900
C08064=1136.455,200.604,-63.647,-178.171,7.548,148.900
C08065=1136.451,200.853,-63.671,-178.169,7.551,148.900
C08066=1136.446,201.102,-63.696,-178.165,7.554,148.899
C08067=1136.442,201.350,-63.721,-178.163,7.557,148.899
C08068=1136.437,201.599,-63.744,-178.160,7.559,148.899
C08069=1136.433,201.849,-63.769,-178.157,7.561,148.899
C08070=1136.428,202.097,-63.793,-178.154,7.564,148.899
C08071=1136.423,202.346,-63.818,-178.152,7.566,148.898
C08072=1136.419,202.595,-63.842,-178.149,7.569,148.898
C08073=1136.414,202.844,-63.867,-178.146,7.572,148.898
C08074=1136.410,203.092,-63.891,-178.143,7.574,148.898
C08075=1136.406,203.341,-63.916,-178.140,7.576,148.898
C08076=1136.401,203.589,-63.941,-178.138,7.579,148.897
C08077=1136.397,203.838,-63.965,-178.135,7.582,148.897
C08078=1136.392,204.087,-63.990,-178.131,7.585,148.897
C08079=1136.388,204.336,-64.014,-178.129,7.587,148.897
C08080=1136.383,204.584,-64.039,-178.126,7.590,148.897
C08081=1136.379,204.834,-64.063,-178.123,7.592,148.896
C08082=1136.374,205.082,-64.088,-178.120,7.595,148.896
C08083=1136.369,205.331,-64.112,-178.118,7.597,148.896
C08084=1136.365,205.580,-64.137,-178.115,7.600,148.896
C08085=1136.360,205.828,-64.162,-178.112,7.602,148.896
C08086=1136.356,206.077,-64.186,-178.109,7.605,148.896
C08087=1136.351,206.326,-64.211,-178.106,7.608,148.895
C08088=1136.347,206.574,-64.235,-178.104,7.610,148.895
C08089=1136.342,206.824,-64.260,-178.101,7.613,148.895
C08090=1136.337,207.072,-64.286,-178.098,7.615,148.895
C08091=1136.333,207.320,-64.310,-178.095,7.618,148.895
C08092=1136.328,207.570,-64.335,-178.093,7.620,148.895
C08093=1136.324,207.818,-64.359,-178.089,7.623,148.894
C08094=1136.320,208.067,-64.385,-178.087,7.626,148.894
C08095=1136.315,208.316,-64.409,-178.084,7.629,148.894
C08096=1136.310,208.564,-64.433,-178.081,7.632,148.894
C08097=1136.306,208.813,-64.459,-178.078,7.633,148.894
C08098=1136.301,209.083,-64.486,-178.075,7.636,148.893
C08099=1136.296,209.354,-64.513,-178.072,7.640,148.893
C08100=1136.291,209.625,-64.541,-178.069,7.643,148.893
C08101=1136.286,209.895,-64.567,-178.066,7.645,148.893
C08102=1136.281,210.145,-64.592,-178.063,7.648,148.893
C08103=1136.277,210.393,-64.617,-178.060,7.650,148.892
C08104=1136.273,210.642,-64.642,-178.058,7.653,148.892
C08105=1136.268,210.890,-64.668,-178.055,7.656,148.892
C08106=1136.264,211.139,-64.692,-178.051,7.658,148.892
C08107=1136.259,211.388,-64.717,-178.049,7.661,148.892
C08108=1136.255,211.637,-64.742,-178.046,7.663,148.892
C08109=1136.250,211.886,-64.767,-178.044,7.666,148.892
C08110=1136.245,212.134,-64.793,-178.040,7.669,148.891
C08111=1136.241,212.383,-64.817,-178.038,7.672,148.891
C08112=1136.237,212.632,-64.843,-178.035,7.675,148.891
C08113=1136.232,212.880,-64.868,-178.032,7.678,148.891
C08114=1136.227,213.129,-64.893,-178.029,7.679,148.891
C08115=1136.223,213.377,-64.919,-178.026,7.682,148.891
C08116=1136.219,213.626,-64.943,-178.024,7.685,148.890
C08117=1136.215,213.875,-64.969,-178.021,7.688,148.890
C08118=1136.209,214.124,-64.993,-178.018,7.691,148.890
C08119=1136.205,214.373,-65.019,-178.015,7.693,148.890
C08120=1136.200,214.621,-65.045,-178.013,7.696,148.890
C08121=1136.196,214.870,-65.070,-178.010,7.698,148.890
C08122=1136.192,215.118,-65.094,-178.007,7.701,148.890
C08123=1136.188,215.367,-65.120,-178.004,7.704,148.889
C08124=1136.183,215.616,-65.145,-178.001,7.707,148.889
C08125=1136.178,215.864,-65.171,-177.998,7.710,148.889
C08126=1136.174,216.113,-65.196,-177.996,7.712,148.889
C08127=1136.169,216.361,-65.222,-177.993,7.715,148.889
C08128=1136.165,216.611,-65.247,-177.990,7.717,148.889
C08129=1136.160,216.859,-65.272,-177.987,7.720,148.888
C08130=1136.156,217.108,-65.298,-177.984,7.723,148.888
C08131=1136.151,217.356,-65.324,-177.981,7.726,148.888
C08132=1136.146,217.605,-65.348,-177.979,7.728,148.888
C08133=1136.142,217.854,-65.374,-177.976,7.731,148.888
C08134=1136.138,218.103,-65.400,-177.973,7.734,148.888
C08135=1136.133,218.351,-65.425,-177.970,7.736,148.888
C08136=1136.129,218.600,-65.451,-177.967,7.739,148.888
C08137=1136.124,218.848,-65.477,-177.965,7.742,148.887
C08138=1136.120,219.096,-65.502,-177.962,7.745,148.887
C08139=1136.115,219.346,-65.527,-177.958,7.748,148.887
C08140=1136.111,219.595,-65.553,-177.956,7.750,148.887
C08141=1136.106,219.843,-65.578,-177.953,7.753,148.887
C08142=1136.102,220.092,-65.604,-177.951,7.756,148.887
C08143=1136.098,220.340,-65.630,-177.948,7.758,148.887
C08144=1136.093,220.589,-65.655,-177.945,7.761,148.887
C08145=1136.089,220.837,-65.681,-177.942,7.764,148.886
C08146=1136.084,221.086,-65.707,-177.939,7.767,148.886
C08147=1136.080,221.335,-65.732,-177.936,7.770,148.886
C08148=1136.075,221.583,-65.758,-177.934,7.772,148.886
C08149=1136.071,221.832,-65.783,-177.931,7.775,148.886
C08150=1136.067,222.081,-65.809,-177.928,7.778,148.886
C08151=1136.062,222.330,-65.836,-177.925,7.781,148.886
C08152=1136.057,222.578,-65.861,-177.922,7.783,148.885
C08153=1136.053,222.827,-65.887,-177.919,7.786,148.885
C08154=1136.049,223.075,-65.912,-177.917,7.789,148.885
C08155=1136.044,223.324,-65.938,-177.914,7.792,148.885
C08156=1136.040,223.572,-65.964,-177.911,7.795,148.885
C08157=1136.035,223.821,-65.991,-177.909,7.797,148.885
C08158=1136.031,224.070,-66.016,-177.906,7.800,148.885
C08159=1136.026,224.318,-66.042,-177.903,7.802,148.884
C08160=1136.022,224.567,-66.068,-177.900,7.805,148.884
C08161=1136.017,224.815,-66.093,-177.897,7.808,148.884
C08162=1136.013,225.064,-66.120,-177.894,7.811,148.884
C08163=1136.008,225.313,-66.146,-177.891,7.814,148.884
C08164=1136.004,225.562,-66.172,-177.889,7.817,148.884
C08165=1135.999,225.810,-66.197,-177.886,7.820,148.884
C08166=1135.994,226.059,-66.224,-177.883,7.823,148.884
C08167=1135.991,226.307,-66.250,-177.880,7.825,148.884
C08168=1135.986,226.556,-66.276,-177.877,7.828,148.884
C08169=1135.982,226.805,-66.302,-177.875,7.830,148.883
C08170=1135.977,227.053,-66.329,-177.872,7.833,148.883
C08171=1135.973,227.301,-66.354,-177.869,7.836,148.883
C08172=1135.968,227.550,-66.380,-177.866,7.839,148.883
C08173=1135.964,227.798,-66.407,-177.863,7.842,148.883
C08174=1135.960,228.047,-66.433,-177.861,7.845,148.883
C08175=1135.955,228.296,-66.458,-177.858,7.848,148.883
C08176=1135.951,228.545,-66.485,-177.855,7.850,148.883
C08177=1135.946,228.793,-66.511,-177.852,7.853,148.883
C08178=1135.942,229.042,-66.538,-177.849,7.856,148.882
C08179=1135.937,229.290,-66.564,-177.847,7.859,148.882
C08180=1135.933,229.539,-66.589,-177.844,7.862,148.882
C08181=1135.928,229.787,-66.616,-177.841,7.865,148.882
C08182=1135.924,230.036,-66.642,-177.838,7.868,148.882
C08183=1135.920,230.284,-66.669,-177.835,7.870,148.882
C08184=1135.915,230.533,-66.695,-177.832,7.873,148.882
C08185=1135.911,230.782,-66.721,-177.830,7.875,148.882
C08186=1135.906,231.031,-66.748,-177.827,7.878,148.881
C08187=1135.902,231.279,-66.774,-177.824,7.881,148.881
C08188=1135.897,231.528,-66.801,-177.821,7.884,148.881
C08189=1135.893,231.776,-66.827,-177.819,7.887,148.881
C08190=1135.889,232.024,-66.854,-177.816,7.890,148.881
C08191=1135.884,232.273,-66.880,-177.813,7.893,148.881
C08192=1135.880,232.522,-66.906,-177.810,7.896,148.881
C08193=1135.875,232.770,-66.932,-177.807,7.899,148.881
C08194=1135.871,233.018,-66.959,-177.805,7.902,148.881
C08195=1135.866,233.267,-66.986,-177.802,7.905,148.881
C08196=1135.861,233.516,-67.012,-177.799,7.907,148.881
C08197=1135.857,233.764,-67.039,-177.796,7.910,148.881
C08198=1135.853,234.012,-67.066,-177.793,7.913,148.880
C08199=1135.849,234.261,-67.091,-177.791,7.916,148.880
C08200=1135.844,234.510,-67.119,-177.788,7.919,148.880
C08201=1135.840,234.758,-67.145,-177.785,7.922,148.880
C08202=1135.835,235.031,-67.174,-177.782,7.925,148.880
C08203=1135.830,235.303,-67.203,-177.778,7.928,148.880
C08204=1135.825,235.575,-67.233,-177.776,7.931,148.880
C08205=1135.821,235.846,-67.262,-177.773,7.934,148.880
C08206=1135.816,236.095,-67.288,-177.770,7.937,148.880
C08207=1135.811,236.344,-67.315,-177.767,7.940,148.880
C08208=1135.808,236.592,-67.342,-177.764,7.943,148.879
C08209=1135.803,236.840,-67.369,-177.762,7.946,148.879
C08210=1135.798,237.089,-67.396,-177.759,7.949,148.879
C08211=1135.794,237.337,-67.422,-177.756,7.952,148.879
C08212=1135.790,237.586,-67.449,-177.753,7.954,148.879
C08213=1135.785,237.835,-67.476,-177.750,7.957,148.879
C08214=1135.781,238.083,-67.502,-177.747,7.960,148.879
C08215=1135.777,238.332,-67.530,-177.745,7.963,148.879
C08216=1135.772,238.581,-67.557,-177.742,7.966,148.879
C08217=1135.768,238.829,-67.583,-177.739,7.969,148.879
C08218=1135.764,239.077,-67.610,-177.736,7.972,148.879
C08219=1135.759,239.326,-67.637,-177.733,7.975,148.879
C08220=1135.754,239.574,-67.664,-177.731,7.978,148.878
C08221=1135.750,239.822,-67.691,-177.728,7.981,148.878
C08222=1135.746,240.071,-67.718,-177.725,7.983,148.878
C08223=1135.741,240.319,-67.745,-177.723,7.987,148.878
C08224=1135.737,240.569,-67.772,-177.720,7.990,148.878
C08225=1135.732,240.817,-67.799,-177.717,7.993,148.878
C08226=1135.728,241.065,-67.826,-177.714,7.995,148.878
C08227=1135.724,241.314,-67.853,-177.711,7.998,148.878
C08228=1135.719,241.562,-67.880,-177.708,8.002,148.878
C08229=1135.715,241.810,-67.908,-177.705,8.005,148.878
C08230=1135.711,242.059,-67.935,-177.702,8.008,148.878
C08231=1135.707,242.308,-67.962,-177.700,8.011,148.878
C08232=1135.702,242.556,-67.989,-177.697,8.014,148.878
C08233=1135.697,242.805,-68.016,-177.694,8.017,148.878
C08234=1135.693,243.053,-68.043,-177.691,8.020,148.878
C08235=1135.689,243.302,-68.071,-177.688,8.022,148.877
C08236=1135.684,243.550,-68.098,-177.686,8.025,148.877
C08237=1135.680,243.799,-68.125,-177.683,8.028,148.877
C08238=1135.675,244.047,-68.152,-177.680,8.031,148.877
C08239=1135.671,244.295,-68.179,-177.677,8.034,148.877
C08240=1135.667,244.544,-68.207,-177.674,8.037,148.877
C08241=1135.663,244.792,-68.234,-177.672,8.040,148.877
C08242=1135.658,245.041,-68.261,-177.669,8.043,148.877
C08243=1135.654,245.289,-68.289,-177.666,8.046,148.877
C08244=1135.650,245.538,-68.316,-177.664,8.049,148.877
C08245=1135.645,245.786,-68.343,-177.661,8.052,148.877
C08246=1135.641,246.034,-68.371,-177.658,8.055,148.877
C08247=1135.636,246.283,-68.398,-177.655,8.058,148.877
C08248=1135.632,246.532,-68.425,-177.652,8.061,148.877
C08249=1135.628,246.780,-68.453,-177.650,8.064,148.877
C08250=1135.623,247.028,-68.480,-177.646,8.067,148.877
C08251=1135.619,247.278,-68.508,-177.643,8.070,148.876
C08252=1135.614,247.525,-68.535,-177.641,8.073,148.877
C08253=1135.610,247.774,-68.563,-177.638,8.076,148.877
C08254=1135.605,248.022,-68.590,-177.636,8.079,148.876
C08255=1135.601,248.271,-68.618,-177.633,8.082,148.876
C08256=1135.597,248.519,-68.645,-177.630,8.085,148.876
C08257=1135.592,248.767,-68.673,-177.627,8.088,148.876
C08258=1135.589,249.016,-68.701,-177.624,8.091,148.876
C08259=1135.583,249.265,-68.728,-177.622,8.094,148.876
C08260=1135.579,249.513,-68.756,-177.619,8.097,148.876
C08261=1135.575,249.762,-68.784,-177.616,8.100,148.876
C08262=1135.571,250.010,-68.811,-177.614,8.103,148.876
C08263=1135.566,250.258,-68.838,-177.611,8.106,148.876
C08264=1135.562,250.507,-68.867,-177.607,8.109,148.876
C08265=1135.558,250.755,-68.894,-177.605,8.112,148.876
C08266=1135.554,251.004,-68.922,-177.602,8.115,148.876
C08267=1135.549,251.252,-68.950,-177.599,8.118,148.876
C08268=1135.544,251.500,-68.978,-177.597,8.121,148.876
C08269=1135.540,251.749,-69.005,-177.594,8.124,148.876
C08270=1135.536,251.997,-69.033,-177.591,8.127,148.876
C08271=1135.532,252.246,-69.061,-177.588,8.130,148.876
C08272=1135.527,252.494,-69.089,-177.585,8.133,148.876
C08273=1135.522,252.742,-69.117,-177.583,8.136,148.876
C08274=1135.519,252.991,-69.145,-177.579,8.140,148.875
C08275=1135.514,253.239,-69.173,-177.577,8.143,148.876
C08276=1135.510,253.488,-69.200,-177.574,8.146,148.876
C08277=1135.505,253.736,-69.228,-177.571,8.149,148.875
C08278=1135.501,253.984,-69.256,-177.568,8.152,148.875
C08279=1135.497,254.232,-69.284,-177.566,8.155,148.875
C08280=1135.492,254.481,-69.312,-177.563,8.158,148.875
C08281=1135.488,254.730,-69.340,-177.561,8.161,148.875
C08282=1135.484,254.978,-69.368,-177.558,8.164,148.875
C08283=1135.480,255.226,-69.396,-177.554,8.167,148.875
C08284=1135.475,255.475,-69.424,-177.552,8.170,148.875
C08285=1135.471,255.723,-69.453,-177.549,8.173,148.875
C08286=1135.467,255.971,-69.480,-177.546,8.177,148.875
C08287=1135.462,256.220,-69.509,-177.544,8.179,148.875
C08288=1135.457,256.468,-69.536,-177.541,8.182,148.875
C08289=1135.454,256.717,-69.564,-177.538,8.185,148.875
C08290=1135.449,256.965,-69.593,-177.535,8.188,148.875
C08291=1135.445,257.214,-69.621,-177.532,8.192,148.875
C08292=1135.440,257.462,-69.649,-177.529,8.195,148.875
C08293=1135.436,257.710,-69.677,-177.527,8.198,148.875
C08294=1135.432,257.958,-69.705,-177.524,8.201,148.875
C08295=1135.427,258.207,-69.734,-177.521,8.204,148.875
C08296=1135.423,258.455,-69.762,-177.519,8.207,148.875
C08297=1135.418,258.704,-69.790,-177.516,8.210,148.875
C08298=1135.414,258.952,-69.818,-177.513,8.213,148.875
C08299=1135.410,259.200,-69.848,-177.510,8.217,148.875
C08300=1135.406,259.449,-69.876,-177.507,8.220,148.875
C08301=1135.402,259.697,-69.903,-177.505,8.223,148.875
C08302=1135.397,259.945,-69.932,-177.502,8.226,148.875
C08303=1135.393,260.193,-69.960,-177.499,8.229,148.875
C08304=1135.388,260.442,-69.989,-177.496,8.232,148.875
C08305=1135.384,260.690,-70.016,-177.493,8.236,148.875
C08306=1135.380,260.964,-70.049,-177.490,8.239,148.875
C08307=1135.375,261.237,-70.080,-177.487,8.242,148.875
C08308=1135.370,261.512,-70.111,-177.484,8.245,148.875
C08309=1135.365,261.785,-70.142,-177.481,8.249,148.875
C08310=1135.361,262.033,-70.171,-177.479,8.252,148.875
C08311=1135.356,262.281,-70.200,-177.476,8.255,148.875
C08312=1135.352,262.530,-70.228,-177.473,8.258,148.875
C08313=1135.348,262.779,-70.257,-177.470,8.262,148.875
C08314=1135.326,264.052,-70.404,-178.378,10.056,149.563
C08315=1135.322,264.300,-70.434,-178.374,10.059,149.563
C08316=1135.318,264.548,-70.463,-178.371,10.062,149.563
C08317=1135.313,264.797,-70.492,-178.369,10.064,149.563
C08318=1135.308,265.045,-70.521,-178.367,10.066,149.562
C08319=1135.304,265.293,-70.550,-178.364,10.068,149.562
C08320=1135.300,265.541,-70.580,-178.362,10.071,149.562
C08321=1135.296,265.790,-70.608,-178.360,10.073,149.562
C08322=1135.292,266.038,-70.637,-178.357,10.075,149.562
C08323=1135.288,266.263,-70.664,-178.354,10.077,149.562
C08324=1135.284,266.487,-70.690,-178.352,10.080,149.562
C08325=1135.280,266.710,-70.716,-178.350,10.082,149.562
C08326=1135.276,266.935,-70.743,-178.348,10.084,149.562
C08327=1135.272,267.159,-70.769,-178.346,10.086,149.562
C08328=1135.268,267.383,-70.795,-178.344,10.088,149.562
C08329=1135.265,267.607,-70.822,-178.341,10.090,149.562
C08330=1135.261,267.832,-70.848,-178.339,10.092,149.562
C08331=1135.256,268.080,-70.878,-178.336,10.095,149.561
C08332=1135.252,268.328,-70.907,-178.334,10.097,149.561
C08333=1135.248,268.576,-70.937,-178.331,10.099,149.561
C08334=1135.243,268.824,-70.966,-178.329,10.102,149.561
C08335=1135.239,269.072,-70.995,-178.326,10.104,149.561
C08336=1135.235,269.320,-71.025,-178.323,10.107,149.561
C08337=1135.231,269.569,-71.054,-178.321,10.109,149.561
C08338=1135.226,269.817,-71.084,-178.318,10.112,149.561
C08339=1135.222,270.065,-71.113,-178.315,10.115,149.561
C08340=1135.218,270.314,-71.143,-178.313,10.117,149.561
C08341=1135.214,270.562,-71.172,-178.310,10.119,149.560
C08342=1135.210,270.810,-71.201,-178.307,10.122,149.560
C08343=1135.206,271.058,-71.231,-178.304,10.125,149.560
C08344=1135.201,271.307,-71.260,-178.301,10.128,149.560
C08345=1135.197,271.554,-71.289,-178.298,10.130,149.560
C08346=1135.192,271.802,-71.319,-178.296,10.132,149.560
C08347=1135.188,272.051,-71.348,-178.293,10.135,149.560
C08348=1135.184,272.299,-71.378,-178.290,10.138,149.560
C08349=1135.180,272.547,-71.407,-178.286,10.140,149.559
C08350=1135.176,272.795,-71.437,-178.283,10.143,149.559
C08351=1135.171,273.044,-71.467,-178.280,10.146,149.559
C08352=1135.167,273.292,-71.497,-178.277,10.149,149.559
C08353=1135.163,273.540,-71.526,-178.275,10.151,149.559
C08354=1135.159,273.788,-71.556,-178.272,10.154,149.559
C08355=1135.154,274.037,-71.585,-178.268,10.157,149.559
C08356=1135.150,274.285,-71.615,-178.265,10.159,149.559
C08357=1135.146,274.532,-71.645,-178.262,10.162,149.558
C08358=1135.141,274.781,-71.675,-178.259,10.165,149.558
C08359=1135.137,275.029,-71.704,-178.255,10.168,149.558
C08360=1135.133,275.278,-71.734,-178.253,10.171,149.558
C08361=1135.129,275.525,-71.764,-178.250,10.174,149.558
C08362=1135.125,275.773,-71.794,-178.246,10.176,149.558
C08363=1135.120,276.022,-71.824,-178.243,10.179,149.557
C08364=1135.117,276.270,-71.854,-178.239,10.182,149.557
C08365=1135.113,276.519,-71.884,-178.236,10.185,149.557
C08366=1135.108,276.767,-71.913,-178.233,10.187,149.557
C08367=1135.104,277.015,-71.944,-178.230,10.190,149.557
C08368=1135.100,277.263,-71.973,-178.227,10.193,149.557
C08369=1135.095,277.511,-72.003,-178.223,10.196,149.556
C08370=1135.092,277.759,-72.033,-178.219,10.199,149.556
C08371=1135.087,278.008,-72.063,-178.216,10.202,149.556
C08372=1135.083,278.255,-72.093,-178.213,10.204,149.556
C08373=1135.079,278.504,-72.123,-178.209,10.208,149.556
C08374=1135.074,278.752,-72.153,-178.206,10.210,149.555
C08375=1135.070,279.000,-72.183,-178.202,10.213,149.555
C08376=1135.067,279.248,-72.213,-178.199,10.216,149.555
C08377=1135.062,279.497,-72.243,-178.195,10.219,149.555
C08378=1135.058,279.744,-72.273,-178.192,10.222,149.554
C08379=1135.054,279.959,-72.300,-178.189,10.224,149.554
C08380=1135.050,280.172,-72.325,-178.185,10.227,149.554
C08381=1135.047,280.387,-72.351,-178.183,10.230,149.554
C08382=1135.043,280.600,-72.377,-178.179,10.232,149.554
C08383=1135.040,280.814,-72.403,-178.176,10.234,149.553
C08384=1135.036,281.028,-72.429,-178.173,10.237,149.553
C08385=1135.032,281.241,-72.456,-178.170,10.240,149.553
C08386=1135.028,281.456,-72.482,-178.167,10.242,149.553
C08387=1135.024,281.704,-72.512,-178.163,10.245,149.553
C08388=1135.020,281.952,-72.542,-178.160,10.248,149.552
C08389=1135.016,282.200,-72.572,-178.157,10.250,149.552
C08390=1135.012,282.448,-72.603,-178.154,10.253,149.552
C08391=1135.008,282.697,-72.633,-178.151,10.255,149.552
C08392=1135.003,282.945,-72.664,-178.148,10.257,149.552
C08393=1134.999,283.192,-72.694,-178.145,10.260,149.552
C08394=1134.994,283.440,-72.724,-178.142,10.262,149.551
C08395=1134.991,283.689,-72.754,-178.139,10.265,149.551
C08396=1134.986,283.937,-72.785,-178.136,10.267,149.551
C08397=1134.982,284.185,-72.815,-178.133,10.270,149.551
C08398=1134.978,284.433,-72.846,-178.130,10.273,149.551
C08399=1134.974,284.681,-72.876,-178.127,10.275,149.550
C08400=1134.970,284.929,-72.907,-178.123,10.278,149.550
C08401=1134.965,285.178,-72.937,-178.120,10.281,149.550
C08402=1134.961,285.425,-72.967,-178.117,10.283,149.550
C08403=1134.957,285.674,-72.999,-178.115,10.285,149.550
C08404=1134.953,285.922,-73.029,-178.112,10.288,149.550
C08405=1134.949,286.170,-73.060,-178.108,10.290,149.549
C08406=1134.944,286.418,-73.090,-178.105,10.293,149.549
C08407=1134.941,286.666,-73.121,-178.102,10.295,149.549
C08408=1134.936,286.914,-73.152,-178.099,10.298,149.549
C08409=1134.932,287.162,-73.182,-178.096,10.300,149.549
C08410=1134.928,287.410,-73.213,-178.093,10.303,149.548
C08411=1134.924,287.658,-73.244,-178.090,10.306,149.548
C08412=1134.920,287.906,-73.274,-178.087,10.308,149.548
C08413=1134.916,288.154,-73.305,-178.084,10.311,149.548
C08414=1134.911,288.402,-73.336,-178.080,10.314,149.548
C08415=1134.906,288.650,-73.366,-178.078,10.316,149.548
C08416=1134.903,288.899,-73.397,-178.075,10.318,149.547
C08417=1134.899,289.147,-73.428,-178.072,10.321,149.547
C08418=1134.894,289.395,-73.459,-178.068,10.323,149.547
C08419=1134.891,289.643,-73.489,-178.065,10.326,149.547
C08420=1134.886,289.890,-73.521,-178.062,10.328,149.547
C08421=1134.882,290.138,-73.551,-178.059,10.331,149.547
C08422=1134.878,290.387,-73.582,-178.056,10.334,149.546
C08423=1134.874,290.635,-73.613,-178.053,10.336,149.546
C08424=1134.870,290.883,-73.644,-178.050,10.339,149.546
C08425=1134.865,291.131,-73.675,-178.047,10.342,149.546
C08426=1134.861,291.379,-73.706,-178.044,10.344,149.546
C08427=1134.857,291.627,-73.737,-178.041,10.346,149.545
C08428=1134.853,291.875,-73.767,-178.038,10.349,149.545
C08429=1134.849,292.123,-73.798,-178.035,10.351,149.545
C08430=1134.845,292.371,-73.830,-178.032,10.354,149.545
C08431=1134.840,292.619,-73.861,-178.028,10.356,149.545
C08432=1134.836,292.867,-73.892,-178.026,10.359,149.545
C08433=1134.831,293.115,-73.923,-178.022,10.361,149.544
C08434=1134.828,293.363,-73.954,-178.019,10.364,149.544
C08435=1134.824,293.577,-73.981,-178.017,10.366,149.544
C08436=1134.820,293.790,-74.008,-178.014,10.369,149.544
C08437=1134.817,294.004,-74.035,-178.011,10.371,149.544
C08438=1134.814,294.218,-74.061,-178.009,10.373,149.544
C08439=1134.810,294.432,-74.088,-178.006,10.375,149.543
C08440=1134.807,294.646,-74.115,-178.003,10.377,149.543
C08441=1134.803,294.859,-74.142,-178.000,10.380,149.543
C08442=1134.800,295.073,-74.169,-177.998,10.382,149.543
C08443=1134.795,295.321,-74.200,-177.995,10.384,149.543
C08444=1134.792,295.569,-74.232,-177.992,10.387,149.543
C08445=1134.787,295.817,-74.262,-177.989,10.389,149.542
C08446=1134.783,296.065,-74.294,-177.986,10.392,149.542
C08447=1134.779,296.313,-74.325,-177.982,10.395,149.542
C08448=1134.775,296.561,-74.357,-177.979,10.397,149.542
C08449=1134.770,296.809,-74.387,-177.976,10.400,149.542
C08450=1134.767,297.057,-74.419,-177.974,10.402,149.542
C08451=1134.762,297.305,-74.450,-177.970,10.404,149.541
C08452=1134.758,297.553,-74.482,-177.967,10.407,149.541
C08453=1134.754,297.801,-74.513,-177.964,10.409,149.541
C08454=1134.750,298.049,-74.545,-177.961,10.412,149.541
C08455=1134.745,298.297,-74.575,-177.958,10.415,149.541
C08456=1134.742,298.545,-74.607,-177.955,10.417,149.540
C08457=1134.737,298.793,-74.639,-177.952,10.420,149.540
C08458=1134.733,299.041,-74.670,-177.949,10.423,149.540
C08459=1134.729,299.289,-74.701,-177.945,10.425,149.540
C08460=1134.725,299.537,-74.734,-177.942,10.428,149.540
C08461=1134.721,299.786,-74.765,-177.939,10.430,149.540
C08462=1134.716,300.033,-74.796,-177.936,10.433,149.539
C08463=1134.713,300.281,-74.828,-177.933,10.435,149.539
C08464=1134.708,300.528,-74.860,-177.930,10.437,149.539
C08465=1134.704,300.777,-74.891,-177.927,10.440,149.539
C08466=1134.701,301.025,-74.923,-177.924,10.442,149.539
C08467=1134.696,301.272,-74.954,-177.921,10.445,149.538
C08468=1134.692,301.521,-74.987,-177.917,10.447,149.538
C08469=1134.687,301.769,-75.017,-177.915,10.450,149.538
C08470=1134.684,302.017,-75.049,-177.911,10.453,149.538
C08471=1134.680,302.265,-75.081,-177.908,10.455,149.538
C08472=1134.676,302.512,-75.112,-177.905,10.458,149.537
C08473=1134.671,302.760,-75.145,-177.902,10.461,149.537
C08474=1134.667,303.008,-75.177,-177.899,10.463,149.537
C08475=1134.663,303.256,-75.208,-177.896,10.466,149.537
C08476=1134.659,303.504,-75.239,-177.892,10.468,149.537
C08477=1134.655,303.753,-75.272,-177.889,10.471,149.537
C08478=1134.650,304.000,-75.303,-177.886,10.473,149.536
C08479=1134.647,304.248,-75.335,-177.883,10.476,149.536
C08480=1134.643,304.496,-75.367,-177.880,10.479,149.536
C08481=1134.638,304.744,-75.399,-177.877,10.480,149.536
C08482=1134.634,304.992,-75.431,-177.874,10.483,149.536
C08483=1134.630,305.240,-75.463,-177.871,10.485,149.535
C08484=1134.625,305.488,-75.495,-177.868,10.488,149.535
C08485=1134.622,305.736,-75.527,-177.865,10.491,149.535
C08486=1134.618,305.984,-75.558,-177.862,10.493,149.535
C08487=1134.613,306.231,-75.591,-177.858,10.496,149.535
C08488=1134.609,306.479,-75.622,-177.855,10.498,149.534
C08489=1134.606,306.727,-75.654,-177.852,10.501,149.534
C08490=1134.601,306.976,-75.687,-177.849,10.503,149.534
C08491=1134.598,307.189,-75.714,-177.846,10.505,149.534
C08492=1134.594,307.402,-75.742,-177.844,10.508,149.534
C08493=1134.591,307.616,-75.769,-177.841,10.510,149.534
C08494=1134.587,307.830,-75.797,-177.838,10.513,149.534
C08495=1134.584,308.043,-75.825,-177.836,10.515,149.534
C08496=1134.580,308.257,-75.852,-177.833,10.516,149.533
C08497=1134.577,308.470,-75.880,-177.830,10.519,149.533
C08498=1134.573,308.684,-75.908,-177.827,10.521,149.533
C08499=1134.569,308.932,-75.940,-177.824,10.523,149.533
C08500=1134.565,309.180,-75.973,-177.821,10.526,149.533
C08501=1134.560,309.428,-76.004,-177.818,10.529,149.532
C08502=1134.556,309.675,-76.037,-177.815,10.531,149.532
C08503=1134.552,309.923,-76.069,-177.812,10.534,149.532
C08504=1134.548,310.172,-76.101,-177.809,10.536,149.532
C08505=1134.545,310.419,-76.134,-177.805,10.539,149.532
C08506=1134.540,310.667,-76.166,-177.802,10.542,149.531
C08507=1134.536,310.915,-76.198,-177.799,10.544,149.531
C08508=1134.532,311.163,-76.231,-177.796,10.547,149.531
C08509=1134.528,311.411,-76.263,-177.793,10.549,149.531
C08510=1134.524,311.659,-76.295,-177.789,10.552,149.531
C08511=1134.520,311.906,-76.328,-177.787,10.554,149.531
C08512=1134.515,312.154,-76.360,-177.784,10.556,149.530
C08513=1134.511,312.402,-76.392,-177.781,10.559,149.530
C08514=1134.507,312.650,-76.425,-177.777,10.561,149.530
C08515=1134.504,312.898,-76.457,-177.774,10.564,149.530
C08516=1134.499,313.145,-76.490,-177.771,10.566,149.530
C08517=1134.495,313.394,-76.522,-177.768,10.569,149.529
C08518=1134.492,313.641,-76.555,-177.765,10.572,149.529
C08519=1134.487,313.889,-76.587,-177.762,10.574,149.529
C08520=1134.483,314.136,-76.620,-177.758,10.577,149.529
C08521=1134.479,314.385,-76.652,-177.755,10.579,149.529
C08522=1134.475,314.632,-76.685,-177.752,10.582,149.528
C08523=1134.471,314.880,-76.717,-177.749,10.585,149.528
C08524=1134.467,315.128,-76.750,-177.746,10.587,149.528
C08525=1134.462,315.377,-76.783,-177.742,10.589,149.528
C08526=1134.459,315.624,-76.815,-177.740,10.592,149.528
C08527=1134.455,315.872,-76.848,-177.736,10.595,149.528
C08528=1134.450,316.120,-76.881,-177.733,10.597,149.527
C08529=1134.447,316.367,-76.913,-177.730,10.600,149.527
C08530=1134.443,316.615,-76.947,-177.727,10.602,149.527
C08531=1134.438,316.864,-76.979,-177.724,10.605,149.527
C08532=1134.435,317.111,-77.012,-177.721,10.607,149.527
C08533=1134.431,317.359,-77.045,-177.718,10.609,149.526
C08534=1134.426,317.607,-77.077,-177.715,10.612,149.526
C08535=1134.422,317.854,-77.110,-177.711,10.614,149.526
C08536=1134.418,318.101,-77.143,-177.708,10.617,149.526
C08537=1134.414,318.349,-77.176,-177.705,10.620,149.526
C08538=1134.410,318.598,-77.208,-177.702,10.622,149.525
C08539=1134.406,318.845,-77.241,-177.698,10.624,149.525
C08540=1134.402,319.093,-77.274,-177.696,10.627,149.525
C08541=1134.398,319.340,-77.307,-177.692,10.630,149.525
C08542=1134.394,319.589,-77.340,-177.689,10.632,149.525
C08543=1134.390,319.837,-77.373,-177.686,10.635,149.525
C08544=1134.386,320.085,-77.406,-177.683,10.637,149.524
C08545=1134.382,320.332,-77.439,-177.680,10.640,149.524
C08546=1134.378,320.580,-77.472,-177.676,10.643,149.524
C08547=1134.374,320.794,-77.500,-177.674,10.644,149.524
C08548=1134.371,321.006,-77.529,-177.671,10.647,149.524
C08549=1134.367,321.220,-77.557,-177.668,10.649,149.524
C08550=1134.364,321.434,-77.586,-177.665,10.651,149.523
C08551=1134.360,321.647,-77.614,-177.663,10.653,149.523
C08552=1134.357,321.861,-77.643,-177.660,10.655,149.523
C08553=1134.354,322.074,-77.671,-177.657,10.658,149.523
C08554=1134.351,322.287,-77.699,-177.655,10.659,149.523
C08555=1134.346,322.535,-77.733,-177.652,10.662,149.522
C08556=1134.342,322.783,-77.766,-177.648,10.665,149.522
C08557=1134.338,323.031,-77.799,-177.645,10.667,149.522
C08558=1134.334,323.278,-77.832,-177.642,10.670,149.522
C08559=1134.330,323.526,-77.865,-177.639,10.672,149.522
C08560=1134.326,323.774,-77.899,-177.635,10.675,149.521
C08561=1134.322,324.022,-77.932,-177.632,10.678,149.521
C08562=1134.318,324.270,-77.965,-177.629,10.680,149.521
C08563=1134.314,324.517,-77.999,-177.626,10.682,149.521
C08564=1134.310,324.765,-78.032,-177.623,10.685,149.521
C08565=1134.306,325.012,-78.065,-177.620,10.688,149.521
C08566=1134.302,325.260,-78.098,-177.616,10.690,149.520
C08567=1134.298,325.508,-78.132,-177.613,10.693,149.520
C08568=1134.294,325.756,-78.165,-177.610,10.695,149.520
C08569=1134.290,326.004,-78.198,-177.607,10.698,149.520
C08570=1134.286,326.251,-78.232,-177.603,10.700,149.519
C08571=1134.282,326.499,-78.265,-177.600,10.703,149.519
C08572=1134.278,326.747,-78.298,-177.597,10.705,149.519
C08573=1134.274,326.994,-78.332,-177.594,10.708,149.519
C08574=1134.271,327.242,-78.366,-177.591,10.710,149.519
C08575=1134.266,327.490,-78.399,-177.588,10.712,149.519
C08576=1134.262,327.738,-78.432,-177.585,10.715,149.518
C08577=1134.258,327.985,-78.467,-177.582,10.717,149.518
C08578=1134.254,328.233,-78.500,-177.579,10.720,149.518
C08579=1134.250,328.481,-78.533,-177.575,10.722,149.518
C08580=1134.246,328.728,-78.567,-177.572,10.725,149.518
C08581=1134.242,328.976,-78.600,-177.569,10.728,149.517
C08582=1134.238,329.224,-78.633,-177.566,10.730,149.517
C08583=1134.233,329.471,-78.668,-177.562,10.733,149.517
C08584=1134.230,329.720,-78.701,-177.559,10.735,149.517
C08585=1134.226,329.967,-78.735,-177.556,10.738,149.517
C08586=1134.222,330.214,-78.768,-177.553,10.740,149.516
C08587=1134.218,330.462,-78.802,-177.549,10.743,149.516
C08588=1134.214,330.710,-78.836,-177.546,10.745,149.516
C08589=1134.210,330.958,-78.870,-177.543,10.748,149.516
C08590=1134.206,331.205,-78.903,-177.540,10.750,149.516
C08591=1134.202,331.453,-78.937,-177.537,10.753,149.515
C08592=1134.198,331.701,-78.971,-177.534,10.756,149.515
C08593=1134.193,331.949,-79.005,-177.530,10.758,149.515
C08594=1134.190,332.196,-79.038,-177.527,10.760,149.515
C08595=1134.186,332.444,-79.073,-177.524,10.763,149.515
C08596=1134.182,332.691,-79.106,-177.521,10.766,149.515
C08597=1134.178,332.939,-79.140,-177.517,10.768,149.514
C08598=1134.174,333.187,-79.174,-177.514,10.771,149.514
C08599=1134.170,333.434,-79.208,-177.511,10.773,149.514
C08600=1134.166,333.682,-79.242,-177.508,10.776,149.514
C08601=1134.162,333.930,-79.276,-177.505,10.778,149.514
C08602=1134.158,334.177,-79.310,-177.501,10.781,149.513
C08603=1134.154,334.391,-79.339,-177.499,10.782,149.513
C08604=1134.151,334.604,-79.368,-177.496,10.784,149.513
C08605=1134.148,334.817,-79.397,-177.493,10.787,149.513
C08606=1134.144,335.031,-79.427,-177.491,10.789,149.513
C08607=1134.141,335.244,-79.456,-177.487,10.791,149.512
C08608=1134.138,335.457,-79.485,-177.485,10.793,149.512
C08609=1134.134,335.670,-79.514,-177.482,10.796,149.512
C08610=1134.131,335.884,-79.545,-177.479,10.798,149.512
C08611=1134.127,336.131,-79.578,-177.476,10.800,149.512
C08612=1134.123,336.379,-79.613,-177.473,10.803,149.511
C08613=1134.119,336.627,-79.646,-177.470,10.805,149.511
C08614=1134.115,336.874,-79.680,-177.467,10.808,149.511
C08615=1134.111,337.122,-79.715,-177.463,10.810,149.511
C08616=1134.107,337.369,-79.749,-177.460,10.813,149.511
C08617=1134.103,337.618,-79.783,-177.457,10.815,149.510
C08618=1134.099,337.865,-79.817,-177.453,10.818,149.510
C08619=1134.095,338.113,-79.852,-177.450,10.821,149.510
C08620=1134.091,338.360,-79.886,-177.447,10.823,149.510
C08621=1134.087,338.607,-79.920,-177.444,10.825,149.510
C08622=1134.083,338.855,-79.954,-177.440,10.828,149.509
C08623=1134.079,339.103,-79.989,-177.437,10.830,149.509
C08624=1134.076,339.350,-80.023,-177.434,10.833,149.509
C08625=1134.071,339.598,-80.058,-177.431,10.836,149.509
C08626=1134.068,339.846,-80.092,-177.428,10.838,149.509
C08627=1134.063,340.093,-80.126,-177.424,10.840,149.508
C08628=1134.059,340.340,-80.161,-177.421,10.843,149.508
C08629=1134.055,340.588,-80.195,-177.418,10.846,149.508
C08630=1134.051,340.836,-80.230,-177.415,10.848,149.508
C08631=1134.048,341.083,-80.264,-177.411,10.851,149.508
C08632=1134.043,341.331,-80.298,-177.409,10.852,149.507
C08633=1134.039,341.579,-80.333,-177.405,10.855,149.507
C08634=1134.035,341.826,-80.367,-177.402,10.857,149.507
C08635=1134.032,342.074,-80.402,-177.399,10.860,149.507
C08636=1134.028,342.321,-80.436,-177.396,10.862,149.507
C08637=1134.024,342.569,-80.471,-177.393,10.865,149.506
C08638=1134.019,342.816,-80.506,-177.389,10.867,149.506
C08639=1134.016,343.064,-80.540,-177.386,10.870,149.506
C08640=1134.011,343.312,-80.574,-177.383,10.872,149.506
C08641=1134.008,343.559,-80.610,-177.380,10.875,149.506
C08642=1134.003,343.806,-80.644,-177.376,10.877,149.505
C08643=1134.000,344.054,-80.679,-177.373,10.880,149.505
C08644=1133.996,344.302,-80.713,-177.370,10.882,149.505
C08645=1133.992,344.549,-80.749,-177.366,10.885,149.505
C08646=1133.989,344.797,-80.783,-177.363,10.887,149.505
C08647=1133.984,345.044,-80.817,-177.360,10.890,149.504
C08648=1133.980,345.292,-80.853,-177.357,10.893,149.504
C08649=1133.976,345.539,-80.887,-177.354,10.895,149.504
C08650=1133.972,345.787,-80.922,-177.350,10.897,149.504
C08651=1133.968,346.034,-80.957,-177.347,10.900,149.504
C08652=1133.964,346.282,-80.992,-177.344,10.902,149.503
C08653=1133.960,346.530,-81.026,-177.340,10.905,149.503
C08654=1133.956,346.777,-81.062,-177.337,10.907,149.503
C08655=1133.953,347.025,-81.096,-177.334,10.910,149.503
C08656=1133.949,347.272,-81.131,-177.331,10.913,149.503
C08657=1133.945,347.520,-81.166,-177.327,10.915,149.502
C08658=1133.941,347.767,-81.201,-177.324,10.917,149.502
C08659=1133.937,347.980,-81.231,-177.321,10.919,149.502
C08660=1133.934,348.193,-81.261,-177.318,10.922,149.502
C08661=1133.931,348.407,-81.291,-177.316,10.924,149.502
C08662=1133.927,348.620,-81.322,-177.313,10.926,149.501
C08663=1133.924,348.833,-81.351,-177.310,10.928,149.501
C08664=1133.920,349.046,-81.381,-177.307,10.931,149.501
C08665=1133.917,349.259,-81.412,-177.304,10.932,149.501
C08666=1133.914,349.473,-81.443,-177.302,10.934,149.501
C08667=1133.910,349.720,-81.476,-177.298,10.937,149.500
C08668=1133.906,349.967,-81.512,-177.294,10.940,149.500
C08669=1133.903,350.215,-81.547,-177.290,10.943,149.500
C08670=1133.898,350.462,-81.582,-177.287,10.945,149.500
C08671=1133.894,350.710,-81.617,-177.283,10.948,149.499
C08672=1133.891,350.957,-81.653,-177.279,10.951,149.499
C08673=1133.887,351.205,-81.688,-177.275,10.954,149.499
C08674=1133.882,351.452,-81.723,-177.272,10.956,149.498
C08675=1133.879,351.700,-81.759,-177.268,10.959,149.498
C08676=1133.875,351.948,-81.793,-177.264,10.962,149.498
C08677=1133.871,352.195,-81.829,-177.261,10.964,149.498
C08678=1133.867,352.442,-81.864,-177.257,10.967,149.497
C08679=1133.863,352.690,-81.900,-177.254,10.970,149.497
C08680=1133.859,352.938,-81.935,-177.249,10.972,149.497
C08681=1133.855,353.184,-81.970,-177.246,10.975,149.497
C08682=1133.851,353.432,-82.005,-177.243,10.977,149.496
C08683=1133.848,353.679,-82.041,-177.238,10.980,149.496
C08684=1133.844,353.927,-82.076,-177.235,10.983,149.496
C08685=1133.840,354.174,-82.112,-177.232,10.985,149.496
C08686=1133.836,354.421,-82.147,-177.228,10.988,149.495
C08687=1133.832,354.669,-82.183,-177.224,10.991,149.495
C08688=1133.828,354.917,-82.218,-177.221,10.993,149.495
C08689=1133.824,355.165,-82.254,-177.217,10.996,149.495
C08690=1133.820,355.412,-82.289,-177.213,10.998,149.494
C08691=1133.816,355.659,-82.324,-177.210,11.001,149.494
C08692=1133.812,355.906,-82.360,-177.206,11.003,149.494
C08693=1133.809,356.154,-82.395,-177.203,11.006,149.493
C08694=1133.805,356.401,-82.431,-177.199,11.009,149.493
C08695=1133.801,356.649,-82.467,-177.195,11.011,149.493
C08696=1133.797,356.897,-82.503,-177.192,11.013,149.492
C08697=1133.793,357.143,-82.539,-177.188,11.016,149.492
C08698=1133.789,357.390,-82.574,-177.185,11.018,149.492
C08699=1133.786,357.638,-82.610,-177.182,11.021,149.492
C08700=1133.782,357.885,-82.645,-177.177,11.024,149.491
C08701=1133.778,358.133,-82.681,-177.174,11.026,149.491
C08702=1133.774,358.381,-82.717,-177.171,11.029,149.491
C08703=1133.770,358.628,-82.752,-177.167,11.031,149.491
C08704=1133.767,358.876,-82.788,-177.164,11.033,149.490
C08705=1133.763,359.123,-82.825,-177.161,11.036,149.490
C08706=1133.758,359.370,-82.860,-177.157,11.038,149.490
C08707=1133.755,359.617,-82.896,-177.154,11.040,149.490
C08708=1133.751,359.865,-82.931,-177.150,11.043,149.489
C08709=1133.747,360.112,-82.968,-177.146,11.046,149.489
C08710=1133.743,360.359,-83.004,-177.143,11.048,149.489
C08711=1133.740,360.607,-83.039,-177.139,11.051,149.489
C08712=1133.735,360.855,-83.075,-177.136,11.053,149.488
C08713=1133.732,361.102,-83.112,-177.133,11.056,149.488
C08714=1133.728,361.349,-83.147,-177.129,11.058,149.488
C08715=1133.725,361.562,-83.178,-177.127,11.060,149.488
C08716=1133.722,361.775,-83.209,-177.123,11.062,149.487
C08717=1133.718,361.988,-83.241,-177.121,11.064,149.487
C08718=1133.715,362.201,-83.271,-177.118,11.066,149.487
C08719=1133.712,362.414,-83.303,-177.115,11.068,149.487
C08720=1133.708,362.627,-83.333,-177.112,11.070,149.486
C08721=1133.705,362.840,-83.364,-177.109,11.072,149.486
C08722=1133.702,363.053,-83.395,-177.106,11.074,149.486
C08723=1133.698,363.300,-83.432,-177.103,11.076,149.486
C08724=1133.694,363.548,-83.467,-177.099,11.079,149.486
C08725=1133.690,363.795,-83.504,-177.096,11.081,149.485
C08726=1133.686,364.043,-83.540,-177.093,11.084,149.485
C08727=1133.683,364.289,-83.576,-177.089,11.086,149.485
C08728=1133.679,364.537,-83.612,-177.086,11.088,149.484
C08729=1133.675,364.784,-83.648,-177.083,11.090,149.484
C08730=1133.671,365.031,-83.685,-177.080,11.093,149.484
C08731=1133.668,365.279,-83.721,-177.077,11.095,149.484
C08732=1133.663,365.526,-83.758,-177.073,11.097,149.484
C08733=1133.660,365.774,-83.793,-177.070,11.100,149.483
C08734=1133.656,366.021,-83.830,-177.067,11.102,149.483
C08735=1133.652,366.268,-83.866,-177.063,11.105,149.483
C08736=1133.648,366.516,-83.903,-177.060,11.106,149.483
C08737=1133.645,366.763,-83.939,-177.057,11.109,149.482
C08738=1133.641,367.011,-83.975,-177.054,11.111,149.482
C08739=1133.637,367.258,-84.012,-177.050,11.114,149.482
C08740=1133.633,367.505,-84.048,-177.047,11.116,149.482
C08741=1133.629,367.753,-84.085,-177.044,11.118,149.481
C08742=1133.626,368.000,-84.121,-177.041,11.120,149.481
C08743=1133.621,368.247,-84.158,-177.038,11.123,149.481
C08744=1133.618,368.494,-84.194,-177.034,11.125,149.481
C08745=1133.614,368.741,-84.230,-177.032,11.127,149.481
C08746=1133.610,368.989,-84.267,-177.029,11.129,149.480
C08747=1133.607,369.236,-84.304,-177.025,11.132,149.480
C08748=1133.603,369.483,-84.340,-177.022,11.134,149.480
C08749=1133.599,369.730,-84.377,-177.019,11.136,149.480
C08750=1133.595,369.978,-84.413,-177.016,11.139,149.479
C08751=1133.591,370.225,-84.450,-177.013,11.141,149.479
C08752=1133.588,370.472,-84.486,-177.010,11.144,149.479
C08753=1133.583,370.719,-84.523,-177.007,11.146,149.479
C08754=1133.580,370.967,-84.560,-177.004,11.148,149.479
C08755=1133.577,371.214,-84.596,-177.000,11.150,149.479
C08756=1133.572,371.461,-84.633,-176.998,11.152,149.478
C08757=1133.568,371.709,-84.670,-176.995,11.155,149.478
C08758=1133.565,371.955,-84.706,-176.991,11.157,149.478
C08759=1133.561,372.203,-84.743,-176.989,11.159,149.478
C08760=1133.557,372.450,-84.780,-176.986,11.162,149.478
C08761=1133.553,372.698,-84.817,-176.983,11.163,149.477
C08762=1133.550,372.945,-84.854,-176.980,11.166,149.477
C08763=1133.546,373.192,-84.890,-176.976,11.168,149.477
C08764=1133.542,373.439,-84.927,-176.974,11.170,149.477
C08765=1133.538,373.687,-84.964,-176.971,11.173,149.477
C08766=1133.535,373.934,-85.001,-176.968,11.174,149.476
C08767=1133.531,374.181,-85.038,-176.965,11.177,149.476
C08768=1133.527,374.428,-85.074,-176.962,11.180,149.476
C08769=1133.523,374.676,-85.112,-176.959,11.181,149.476
C08770=1133.519,374.923,-85.149,-176.956,11.184,149.476
C08771=1133.516,375.136,-85.180,-176.954,11.186,149.476
C08772=1133.512,375.349,-85.212,-176.951,11.188,149.476
C08773=1133.510,375.561,-85.244,-176.949,11.190,149.475
C08774=1133.506,375.774,-85.276,-176.946,11.192,149.475
C08775=1133.503,375.987,-85.307,-176.944,11.194,149.475
C08776=1133.500,376.200,-85.339,-176.942,11.195,149.475
C08777=1133.497,376.412,-85.371,-176.939,11.197,149.475
C08778=1133.493,376.625,-85.403,-176.937,11.199,149.475
C08779=1133.490,376.873,-85.440,-176.934,11.202,149.475
C08780=1133.485,377.120,-85.477,-176.931,11.204,149.475
C08781=1133.482,377.367,-85.513,-176.928,11.206,149.474
C08782=1133.479,377.614,-85.551,-176.926,11.208,149.474
C08783=1133.475,377.862,-85.588,-176.923,11.211,149.474
C08784=1133.471,378.109,-85.625,-176.920,11.213,149.474
C08785=1133.467,378.356,-85.662,-176.917,11.215,149.474
C08786=1133.463,378.603,-85.700,-176.915,11.218,149.474
C08787=1133.459,378.850,-85.737,-176.911,11.220,149.474
C08788=1133.455,379.098,-85.773,-176.909,11.222,149.474
C08789=1133.452,379.345,-85.811,-176.906,11.225,149.474
C08790=1133.448,379.592,-85.848,-176.904,11.227,149.473
C08791=1133.444,379.839,-85.885,-176.901,11.229,149.473
C08792=1133.441,380.086,-85.923,-176.898,11.231,149.473
C08793=1133.437,380.334,-85.960,-176.896,11.233,149.473
C08794=1133.433,380.580,-85.997,-176.893,11.236,149.473
C08795=1133.429,380.828,-86.035,-176.891,11.238,149.473
C08796=1133.425,381.075,-86.072,-176.888,11.241,149.473
C08797=1133.421,381.322,-86.109,-176.885,11.243,149.473
C08798=1133.418,381.570,-86.146,-176.882,11.245,149.473
C08799=1133.414,381.816,-86.184,-176.880,11.247,149.473
C08800=1133.410,382.064,-86.221,-176.878,11.249,149.473
C08801=1133.407,382.311,-86.259,-176.875,11.252,149.473
C08802=1133.403,382.558,-86.296,-176.872,11.254,149.473
C08803=1133.400,382.805,-86.334,-176.870,11.256,149.473
C08804=1133.396,383.052,-86.370,-176.867,11.259,149.472
C08805=1133.392,383.299,-86.408,-176.865,11.261,149.472
C08806=1133.388,383.547,-86.445,-176.863,11.263,149.473
C08807=1133.384,383.794,-86.483,-176.862,11.265,149.473
C08808=1133.381,384.041,-86.520,-176.861,11.266,149.473
C08809=1133.377,384.288,-86.558,-176.860,11.267,149.473
C08810=1133.373,384.535,-86.594,-176.859,11.269,149.473
C08811=1133.370,384.782,-86.632,-176.858,11.271,149.473
C08812=1133.366,385.029,-86.670,-176.857,11.272,149.473
C08813=1133.362,385.277,-86.708,-176.855,11.274,149.473
C08814=1133.358,385.524,-86.745,-176.854,11.276,149.474
C08815=1133.354,385.771,-86.782,-176.853,11.277,149.474
C08816=1133.351,386.018,-86.820,-176.852,11.279,149.474
C08817=1133.347,386.265,-86.858,-176.851,11.281,149.474
C08818=1133.344,386.513,-86.895,-176.851,11.282,149.474
C08819=1133.340,386.759,-86.932,-176.850,11.284,149.474
C08820=1133.336,387.007,-86.970,-176.849,11.285,149.475
C08821=1133.332,387.254,-87.007,-176.848,11.287,149.475
C08822=1133.329,387.500,-87.045,-176.847,11.289,149.475
C08823=1133.324,387.749,-87.083,-176.846,11.291,149.475
C08824=1133.321,387.995,-87.120,-176.845,11.293,149.476
C08825=1133.317,388.242,-87.158,-176.844,11.295,149.476
C08826=1133.313,388.490,-87.195,-176.843,11.297,149.476
C08827=1133.310,388.703,-87.228,-176.843,11.298,149.476
C08828=1133.307,388.915,-87.261,-176.842,11.300,149.477
C08829=1133.304,389.128,-87.292,-176.841,11.301,149.477
C08830=1133.301,389.341,-87.325,-176.841,11.303,149.477
C08831=1133.298,389.553,-87.357,-176.840,11.304,149.477
C08832=1133.294,389.765,-87.390,-176.840,11.306,149.478
C08833=1133.292,389.979,-87.422,-176.839,11.307,149.478
C08834=1133.288,390.191,-87.454,-176.838,11.309,149.478
C08835=1133.284,390.438,-87.492,-176.838,11.312,149.479
C08836=1133.280,390.686,-87.530,-176.837,11.313,149.479
C08837=1133.276,390.932,-87.567,-176.837,11.315,149.479
C08838=1133.273,391.180,-87.605,-176.836,11.317,149.480
C08839=1133.269,391.426,-87.643,-176.836,11.319,149.480
C08840=1133.266,391.674,-87.680,-176.835,11.321,149.480
C08841=1133.262,391.921,-87.717,-176.834,11.323,149.481
C08842=1133.258,392.168,-87.756,-176.834,11.325,149.481
C08843=1133.254,392.415,-87.794,-176.833,11.327,149.482
C08844=1133.251,392.663,-87.831,-176.833,11.330,149.482
C08845=1133.247,392.909,-87.868,-176.832,11.332,149.482
C08846=1133.244,393.157,-87.906,-176.832,11.334,149.483
C08847=1133.240,393.403,-87.944,-176.831,11.336,149.483
C08848=1133.236,393.651,-87.982,-176.831,11.338,149.484
C08849=1133.232,393.898,-88.019,-176.830,11.341,149.484
C08850=1133.229,394.145,-88.057,-176.830,11.343,149.485
C08851=1133.225,394.392,-88.095,-176.829,11.345,149.485
C08852=1133.221,394.639,-88.133,-176.830,11.347,149.486
C08853=1133.217,394.887,-88.170,-176.830,11.349,149.486
C08854=1133.213,395.133,-88.208,-176.829,11.351,149.487
C08855=1133.210,395.380,-88.246,-176.829,11.354,149.487
C08856=1133.206,395.627,-88.284,-176.829,11.356,149.488
C08857=1133.202,395.875,-88.322,-176.828,11.358,149.488
C08858=1133.198,396.122,-88.359,-176.828,11.361,149.489
C08859=1133.195,396.369,-88.397,-176.828,11.364,149.490
C08860=1133.191,396.616,-88.435,-176.828,11.366,149.490
C08861=1133.187,396.863,-88.473,-176.827,11.368,149.491
C08862=1133.184,397.110,-88.510,-176.827,11.371,149.491
C08863=1133.180,397.357,-88.548,-176.827,11.373,149.492
C08864=1133.176,397.604,-88.586,-176.827,11.376,149.493
C08865=1133.172,397.852,-88.624,-176.827,11.378,149.493
C08866=1133.169,398.098,-88.661,-176.827,11.381,149.494
C08867=1133.165,398.346,-88.699,-176.827,11.384,149.495
C08868=1133.162,398.593,-88.738,-176.827,11.386,149.495
C08869=1133.158,398.840,-88.775,-176.827,11.389,149.496
C08870=1133.155,399.087,-88.813,-176.827,11.391,149.497
C08871=1133.151,399.334,-88.851,-176.827,11.394,149.497
C08872=1133.147,399.582,-88.889,-176.827,11.397,149.498
C08873=1133.143,399.828,-88.926,-176.827,11.399,149.499
C08874=1133.140,400.076,-88.964,-176.827,11.402,149.499
C08875=1133.135,400.322,-89.002,-176.827,11.405,149.500
C08876=1133.132,400.570,-89.040,-176.828,11.408,149.501
C08877=1133.128,400.816,-89.078,-176.828,11.411,149.502
C08878=1133.125,401.064,-89.116,-176.827,11.414,149.502
C08879=1133.120,401.310,-89.154,-176.827,11.417,149.503
C08880=1133.117,401.558,-89.192,-176.828,11.420,149.504
C08881=1133.113,401.804,-89.229,-176.828,11.423,149.505
C08882=1133.109,402.052,-89.268,-176.828,11.425,149.506
C08883=1133.106,402.264,-89.301,-176.828,11.428,149.506
C08884=1133.104,402.477,-89.333,-176.829,11.430,149.507
C08885=1133.100,402.689,-89.365,-176.829,11.433,149.508
C08886=1133.097,402.902,-89.397,-176.830,11.436,149.509
C08887=1133.094,403.115,-89.430,-176.830,11.438,149.510
C08888=1133.090,403.328,-89.463,-176.830,11.441,149.510
C08889=1133.087,403.541,-89.496,-176.831,11.443,149.511
C08890=1133.084,403.753,-89.528,-176.831,11.446,149.512
C08891=1133.081,404.000,-89.566,-176.832,11.449,149.513
C08892=1133.076,404.247,-89.605,-176.831,11.453,149.514
C08893=1133.073,404.495,-89.642,-176.832,11.456,149.515
C08894=1133.069,404.741,-89.680,-176.832,11.459,149.516
C08895=1133.065,404.989,-89.719,-176.833,11.462,149.517
C08896=1133.061,405.235,-89.756,-176.834,11.465,149.518
C08897=1133.058,405.482,-89.794,-176.835,11.469,149.519
C08898=1133.054,405.730,-89.833,-176.835,11.472,149.520
C08899=1133.051,405.977,-89.870,-176.835,11.476,149.521
C08900=1133.047,406.224,-89.908,-176.836,11.479,149.522
C08901=1133.043,406.471,-89.946,-176.837,11.482,149.523
C08902=1133.040,406.718,-89.984,-176.838,11.485,149.524
C08903=1133.036,406.965,-90.022,-176.839,11.489,149.525
C08904=1133.032,407.212,-90.060,-176.839,11.493,149.526
C08905=1133.029,407.460,-90.098,-176.839,11.496,149.527
C08906=1133.025,407.706,-90.136,-176.840,11.500,149.528
C08907=1133.021,407.954,-90.174,-176.841,11.503,149.529
C08908=1133.018,408.200,-90.213,-176.842,11.507,149.530
C08909=1133.014,408.447,-90.251,-176.843,11.511,149.532
C08910=1133.010,408.694,-90.289,-176.843,11.514,149.533
C08911=1133.007,408.941,-90.327,-176.845,11.518,149.534
C08912=1133.003,409.189,-90.365,-176.846,11.521,149.535
C08913=1132.999,409.435,-90.403,-176.846,11.525,149.536
C08914=1132.996,409.682,-90.441,-176.847,11.529,149.537
C08915=1132.991,409.929,-90.479,-176.848,11.533,149.539
C08916=1132.988,410.177,-90.517,-176.849,11.537,149.540
C08917=1132.985,410.424,-90.555,-176.850,11.541,149.541
C08918=1132.980,410.671,-90.593,-176.851,11.544,149.542
C08919=1132.977,410.918,-90.631,-176.852,11.549,149.544
C08920=1132.973,411.165,-90.669,-176.853,11.553,149.545
C08921=1132.969,411.412,-90.707,-176.855,11.556,149.546
C08922=1132.966,411.658,-90.745,-176.855,11.561,149.548
C08923=1132.962,411.906,-90.784,-176.857,11.565,149.549
C08924=1132.959,412.153,-90.822,-176.858,11.568,149.550
C08925=1132.954,412.400,-90.860,-176.859,11.573,149.552
C08926=1132.951,412.647,-90.898,-176.860,11.577,149.553
C08927=1132.947,412.894,-90.936,-176.862,11.581,149.555
C08928=1132.943,413.141,-90.974,-176.863,11.586,149.556
C08929=1132.940,413.389,-91.012,-176.864,11.589,149.557
C08930=1132.936,413.635,-91.050,-176.865,11.594,149.559
C08931=1132.933,413.882,-91.089,-176.867,11.598,149.560
C08932=1132.929,414.130,-91.127,-176.868,11.602,149.562
C08933=1132.925,414.376,-91.165,-176.869,11.607,149.563
C08934=1132.923,414.624,-91.203,-176.871,11.611,149.565
C08935=1132.921,414.870,-91.241,-176.872,11.616,149.566
C08936=1132.919,415.118,-91.278,-176.874,11.620,149.568
C08937=1132.918,415.365,-91.316,-176.876,11.624,149.569
C08938=1132.918,415.612,-91.354,-176.877,11.629,149.571
C08939=1132.919,415.824,-91.387,-176.878,11.633,149.572
C08940=1132.919,416.036,-91.419,-176.880,11.637,149.574
C08941=1132.920,416.249,-91.451,-176.881,11.641,149.575
C08942=1132.922,416.462,-91.483,-176.883,11.645,149.576
C08943=1132.924,416.674,-91.515,-176.884,11.648,149.578
C08944=1132.926,416.887,-91.547,-176.886,11.652,149.579
C08945=1132.930,417.100,-91.579,-176.887,11.656,149.581
C08946=1132.933,417.312,-91.611,-176.889,11.660,149.582
C08947=1132.514,417.311,-91.673,-176.881,11.665,149.581
C08948=1132.510,417.099,-91.642,-176.879,11.661,149.580
C08949=1132.508,416.887,-91.610,-176.878,11.657,149.578
C08950=1132.505,416.674,-91.578,-176.877,11.653,149.577
C08951=1132.503,416.462,-91.546,-176.875,11.649,149.576
C08952=1132.501,416.249,-91.514,-176.874,11.645,149.574
C08953=1132.500,416.037,-91.481,-176.872,11.641,149.573
C08954=1132.499,415.825,-91.449,-176.871,11.637,149.572
C08955=1132.499,415.611,-91.417,-176.869,11.633,149.570
C08956=1132.500,415.365,-91.379,-176.868,11.628,149.569
C08957=1132.500,415.117,-91.341,-176.867,11.624,149.567
C08958=1132.502,414.871,-91.303,-176.866,11.619,149.566
C08959=1132.504,414.623,-91.265,-176.864,11.615,149.564
C08960=1132.506,414.376,-91.228,-176.863,11.611,149.563
C08961=1132.509,414.130,-91.189,-176.861,11.606,149.561
C08962=1132.513,413.882,-91.150,-176.860,11.602,149.560
C08963=1132.517,413.635,-91.113,-176.859,11.598,149.558
C08964=1132.521,413.388,-91.074,-176.858,11.593,149.557
C08965=1132.525,413.141,-91.037,-176.856,11.589,149.555
C08966=1132.528,412.894,-90.998,-176.856,11.585,149.554
C08967=1132.531,412.647,-90.960,-176.854,11.581,149.553
C08968=1132.535,412.400,-90.922,-176.853,11.577,149.551
C08969=1132.539,412.153,-90.883,-176.852,11.572,149.550
C08970=1132.542,411.906,-90.846,-176.850,11.568,149.548
C08971=1132.547,411.659,-90.807,-176.849,11.564,149.547
C08972=1132.550,411.411,-90.769,-176.848,11.560,149.546
C08973=1132.554,411.165,-90.732,-176.848,11.556,149.544
C08974=1132.558,410.917,-90.693,-176.846,11.552,149.543
C08975=1132.561,410.671,-90.655,-176.845,11.548,149.542
C08976=1132.565,410.424,-90.617,-176.844,11.544,149.541
C08977=1132.568,410.176,-90.579,-176.843,11.540,149.539
C08978=1132.572,409.930,-90.541,-176.842,11.537,149.538
C08979=1132.576,409.682,-90.502,-176.842,11.532,149.537
C08980=1132.579,409.435,-90.465,-176.841,11.529,149.536
C08981=1132.584,409.188,-90.426,-176.840,11.525,149.535
C08982=1132.587,408.941,-90.388,-176.839,11.521,149.533
C08983=1132.591,408.694,-90.351,-176.838,11.517,149.532
C08984=1132.595,408.447,-90.312,-176.837,11.514,149.531
C08985=1132.598,408.199,-90.274,-176.837,11.510,149.530
C08986=1132.602,407.953,-90.236,-176.836,11.506,149.529
C08987=1132.605,407.706,-90.198,-176.835,11.503,149.528
C08988=1132.609,407.459,-90.160,-176.835,11.499,149.526
C08989=1132.613,407.212,-90.121,-176.834,11.496,149.525
C08990=1132.617,406.965,-90.084,-176.833,11.492,149.524
C08991=1132.620,406.718,-90.046,-176.832,11.489,149.523
C08992=1132.624,406.470,-90.007,-176.832,11.485,149.522
C08993=1132.628,406.224,-89.970,-176.831,11.482,149.521
C08994=1132.631,405.977,-89.932,-176.831,11.478,149.520
C08995=1132.635,405.730,-89.894,-176.830,11.475,149.519
C08996=1132.638,405.482,-89.856,-176.830,11.471,149.518
C08997=1132.642,405.235,-89.817,-176.829,11.468,149.517
C08998=1132.646,404.988,-89.780,-176.828,11.465,149.516
C08999=1132.649,404.741,-89.742,-176.828,11.462,149.515
C09000=1132.654,404.494,-89.704,-176.827,11.459,149.514
C09001=1132.657,404.247,-89.666,-176.828,11.455,149.513
C09002=1132.661,404.000,-89.628,-176.827,11.452,149.512
C09003=1132.665,403.753,-89.589,-176.827,11.449,149.511
C09004=1132.668,403.541,-89.557,-176.826,11.446,149.511
C09005=1132.670,403.328,-89.525,-176.826,11.443,149.510
C09006=1132.674,403.115,-89.492,-176.825,11.441,149.509
C09007=1132.677,402.903,-89.459,-176.825,11.438,149.508
C09008=1132.680,402.690,-89.426,-176.825,11.436,149.508
C09009=1132.684,402.478,-89.394,-176.825,11.433,149.507
C09010=1132.687,402.264,-89.361,-176.825,11.430,149.506
C09011=1132.690,402.052,-89.328,-176.825,11.428,149.505
C09012=1132.694,401.806,-89.291,-176.824,11.425,149.505
C09013=1132.697,401.558,-89.253,-176.824,11.422,149.504
C09014=1132.701,401.311,-89.214,-176.824,11.419,149.503
C09015=1132.705,401.064,-89.177,-176.823,11.416,149.502
C09016=1132.708,400.817,-89.139,-176.824,11.413,149.501
C09017=1132.712,400.570,-89.101,-176.823,11.411,149.501
C09018=1132.716,400.322,-89.063,-176.824,11.407,149.500
C09019=1132.720,400.076,-89.026,-176.824,11.404,149.499
C09020=1132.724,399.828,-88.987,-176.823,11.401,149.498
C09021=1132.727,399.581,-88.950,-176.823,11.399,149.498
C09022=1132.731,399.334,-88.912,-176.823,11.396,149.497
C09023=1132.734,399.088,-88.874,-176.823,11.393,149.496
C09024=1132.738,398.840,-88.836,-176.823,11.391,149.495
C09025=1132.742,398.593,-88.798,-176.823,11.388,149.495
C09026=1132.745,398.346,-88.760,-176.823,11.386,149.494
C09027=1132.749,398.100,-88.723,-176.823,11.383,149.494
C09028=1132.753,397.851,-88.685,-176.823,11.381,149.493
C09029=1132.757,397.605,-88.647,-176.824,11.378,149.492
C09030=1132.760,397.357,-88.609,-176.824,11.376,149.492
C09031=1132.765,397.111,-88.571,-176.824,11.373,149.491
C09032=1132.768,396.863,-88.533,-176.824,11.371,149.491
C09033=1132.771,396.616,-88.495,-176.824,11.368,149.490
C09034=1132.775,396.370,-88.458,-176.824,11.366,149.489
C09035=1132.779,396.122,-88.419,-176.825,11.363,149.489
C09036=1132.783,395.875,-88.382,-176.825,11.360,149.488
C09037=1132.786,395.627,-88.344,-176.826,11.358,149.488
C09038=1132.790,395.381,-88.307,-176.826,11.355,149.487
C09039=1132.794,395.133,-88.268,-176.826,11.353,149.487
C09040=1132.798,394.887,-88.231,-176.827,11.351,149.486
C09041=1132.802,394.640,-88.194,-176.827,11.348,149.485
C09042=1132.805,394.392,-88.156,-176.827,11.346,149.485
C09043=1132.810,394.145,-88.118,-176.828,11.344,149.484
C09044=1132.813,393.898,-88.080,-176.828,11.342,149.484
C09045=1132.817,393.652,-88.042,-176.829,11.339,149.484
C09046=1132.820,393.404,-88.005,-176.829,11.337,149.483
C09047=1132.824,393.157,-87.967,-176.829,11.336,149.483
C09048=1132.828,392.910,-87.929,-176.830,11.333,149.482
C09049=1132.832,392.663,-87.891,-176.830,11.331,149.482
C09050=1132.835,392.416,-87.853,-176.830,11.329,149.481
C09051=1132.839,392.168,-87.816,-176.831,11.327,149.481
C09052=1132.842,391.921,-87.778,-176.832,11.325,149.481
C09053=1132.847,391.674,-87.740,-176.832,11.323,149.480
C09054=1132.850,391.427,-87.702,-176.833,11.321,149.480
C09055=1132.854,391.180,-87.665,-176.834,11.319,149.479
C09056=1132.857,390.933,-87.628,-176.834,11.317,149.479
C09057=1132.861,390.686,-87.590,-176.835,11.314,149.479
C09058=1132.864,390.438,-87.553,-176.836,11.313,149.478
C09059=1132.869,390.191,-87.515,-176.837,11.311,149.478
C09060=1132.872,389.979,-87.483,-176.837,11.309,149.478
C09061=1132.874,389.766,-87.450,-176.838,11.308,149.478
C09062=1132.878,389.553,-87.418,-176.839,11.306,149.477
C09063=1132.882,389.341,-87.385,-176.839,11.304,149.477
C09064=1132.884,389.128,-87.353,-176.840,11.303,149.477
C09065=1132.887,388.916,-87.320,-176.840,11.301,149.477
C09066=1132.891,388.703,-87.288,-176.841,11.299,149.476
C09067=1132.894,388.490,-87.255,-176.842,11.298,149.476
C09068=1132.898,388.243,-87.218,-176.842,11.296,149.476
C09069=1132.901,387.995,-87.181,-176.843,11.294,149.475
C09070=1132.905,387.749,-87.143,-176.844,11.292,149.475
C09071=1132.908,387.501,-87.105,-176.845,11.290,149.475
C09072=1132.912,387.254,-87.068,-176.846,11.289,149.475
C09073=1132.916,387.008,-87.031,-176.847,11.287,149.475
C09074=1132.920,386.760,-86.992,-176.848,11.285,149.474
C09075=1132.924,386.513,-86.955,-176.849,11.283,149.474
C09076=1132.927,386.266,-86.917,-176.850,11.281,149.474
C09077=1132.931,386.018,-86.880,-176.851,11.280,149.474
C09078=1132.935,385.771,-86.843,-176.852,11.278,149.474
C09079=1132.938,385.525,-86.805,-176.853,11.276,149.473
C09080=1132.942,385.277,-86.768,-176.854,11.274,149.473
C09081=1132.946,385.030,-86.730,-176.855,11.274,149.473
C09082=1132.950,384.783,-86.693,-176.856,11.272,149.473
C09083=1132.953,384.536,-86.655,-176.857,11.270,149.473
C09084=1132.957,384.289,-86.617,-176.858,11.269,149.473
C09085=1132.962,384.042,-86.580,-176.860,11.267,149.473
C09086=1132.965,383.794,-86.542,-176.861,11.265,149.473
C09087=1132.969,383.547,-86.506,-176.862,11.264,149.472
C09088=1132.972,383.300,-86.468,-176.864,11.261,149.472
C09089=1132.976,383.053,-86.431,-176.866,11.259,149.472
C09090=1132.980,382.806,-86.393,-176.868,11.257,149.472
C09091=1132.983,382.558,-86.356,-176.871,11.255,149.472
C09092=1132.987,382.312,-86.318,-176.874,11.253,149.472
C09093=1132.991,382.064,-86.281,-176.876,11.250,149.472
C09094=1132.994,381.817,-86.244,-176.879,11.248,149.473
C09095=1132.999,381.570,-86.207,-176.881,11.246,149.473
C09096=1133.002,381.323,-86.169,-176.884,11.243,149.473
C09097=1133.006,381.076,-86.132,-176.887,11.241,149.473
C09098=1133.010,380.829,-86.094,-176.890,11.238,149.473
C09099=1133.013,380.581,-86.057,-176.892,11.237,149.473
C09100=1133.017,380.334,-86.020,-176.895,11.234,149.473
C09101=1133.021,380.087,-85.983,-176.897,11.232,149.473
C09102=1133.024,379.839,-85.945,-176.900,11.229,149.473
C09103=1133.029,379.592,-85.909,-176.903,11.227,149.473
C09104=1133.032,379.346,-85.871,-176.905,11.225,149.473
C09105=1133.036,379.098,-85.834,-176.908,11.222,149.473
C09106=1133.040,378.851,-85.797,-176.911,11.221,149.474
